Yaskawa INFORM job: DPRINT3D15.JBI

/JOB
//NAME DPRINT3D15
//POS
///NPOS 1161,0,0,0,0,0
///TOOL 9
///POSTYPE PULSE
///PULSE
C00000=36278,44575,-115468,79318,-120327,-85510,0
C00001=35662,44969,-114487,80045,-120135,-85172,0
C00002=36536,45454,-113310,79361,-120907,-84970,0
C00003=42251,40475,-125838,71885,-121337,-89052,0
C00004=39883,39258,-128907,73938,-119379,-89536,0
C00005=34290,44258,-116221,81147,-118965,-85469,0
C00006=35192,44719,-115096,80418,-119728,-85276,0
C00007=34956,44981,-114446,80729,-119702,-85074,0
C00008=35425,45232,-113838,80359,-120109,-84970,0
C00009=35608,45029,-114339,80116,-120129,-85126,0
C00010=36169,44682,-115203,79459,-120311,-85426,0
C00011=36133,44092,-116660,79301,-120005,-85809,0
C00012=40210,40493,-125752,74007,-120311,-88747,0
C00013=40210,40434,-125759,74020,-120337,-88719,0
C00014=36356,44563,-115373,79269,-120414,-85467,0
C00015=41022,40463,-125699,73192,-120772,-88813,0
C00016=40015,39945,-127000,74059,-119937,-89019,0
C00017=35392,44052,-116619,80042,-119585,-85678,0
C00018=36278,44521,-115476,79331,-120346,-85484,0
C00019=35662,44916,-114494,80057,-120153,-85146,0
C00020=36536,45401,-113317,79374,-120926,-84945,0
C00021=42251,40415,-125845,71899,-121365,-89025,0
C00022=39883,39197,-128913,73951,-119406,-89507,0
C00023=34290,44203,-116228,81159,-118982,-85443,0
C00024=35192,44665,-115103,80431,-119747,-85250,0
C00025=34956,44928,-114453,80742,-119720,-85049,0
C00026=35425,45178,-113845,80371,-120127,-84944,0
C00027=35608,44975,-114347,80129,-120148,-85100,0
C00028=36169,44628,-115210,79472,-120330,-85400,0
C00029=36133,44037,-116667,79314,-120025,-85783,0
C00030=40210,40434,-125759,74020,-120337,-88719,0
C00031=40211,40374,-125767,74034,-120363,-88691,0
C00032=36356,44509,-115380,79282,-120434,-85441,0
C00033=41022,40404,-125706,73206,-120798,-88785,0
C00034=40015,39885,-127008,74073,-119963,-88991,0
C00035=35393,43998,-116625,80054,-119604,-85652,0
C00036=36278,44467,-115483,79344,-120365,-85458,0
C00037=35663,44862,-114501,80070,-120172,-85120,0
C00038=36536,45348,-113324,79387,-120945,-84919,0
C00039=42252,40355,-125852,71914,-121393,-88997,0
C00040=39884,39135,-128921,73965,-119433,-89478,0
C00041=34290,44149,-116235,81171,-119001,-85416,0
C00042=35193,44611,-115110,80443,-119765,-85224,0
C00043=34957,44874,-114460,80754,-119739,-85022,0
C00044=35425,45125,-113852,80384,-120145,-84918,0
C00045=35608,44922,-114354,80141,-120166,-85074,0
C00046=36170,44574,-115218,79485,-120350,-85374,0
C00047=36133,43983,-116674,79327,-120044,-85756,0
C00048=40211,40374,-125767,74034,-120363,-88691,0
C00049=40211,40315,-125774,74048,-120389,-88662,0
C00050=36357,44456,-115387,79295,-120452,-85415,0
C00051=41022,40345,-125714,73220,-120825,-88758,0
C00052=40016,39824,-127015,74086,-119989,-88962,0
C00053=35393,43943,-116632,80066,-119622,-85625,0
C00054=36279,44413,-115490,79356,-120384,-85432,0
C00055=35663,44809,-114508,80082,-120190,-85094,0
C00056=36537,45295,-113331,79400,-120964,-84894,0
C00057=42252,40296,-125860,71928,-121421,-88969,0
C00058=39884,39074,-128928,73978,-119459,-89449,0
C00059=34291,44095,-116242,81183,-119019,-85390,0
C00060=35193,44558,-115117,80455,-119783,-85198,0
C00061=34957,44821,-114467,80766,-119756,-84996,0
C00062=35426,45072,-113859,80396,-120164,-84892,0
C00063=35609,44869,-114361,80154,-120184,-85048,0
C00064=36170,44520,-115225,79497,-120369,-85348,0
C00065=36134,43928,-116681,79339,-120064,-85730,0
C00066=40211,40315,-125774,74048,-120389,-88662,0
C00067=40212,40255,-125781,74062,-120414,-88635,0
C00068=36357,44402,-115394,79307,-120472,-85389,0
C00069=41023,40285,-125721,73234,-120851,-88730,0
C00070=40016,39764,-127022,74100,-120016,-88934,0
C00071=35393,43889,-116639,80079,-119642,-85599,0
C00072=36279,44359,-115497,79369,-120404,-85406,0
C00073=35663,44755,-114514,80095,-120210,-85068,0
C00074=36537,45242,-113338,79413,-120983,-84867,0
C00075=42253,40236,-125867,71943,-121449,-88942,0
C00076=39884,39012,-128936,73992,-119487,-89420,0
C00077=34291,44040,-116249,81195,-119038,-85364,0
C00078=35193,44504,-115124,80468,-119802,-85172,0
C00079=34958,44768,-114474,80779,-119774,-84970,0
C00080=35426,45019,-113866,80409,-120181,-84866,0
C00081=35609,44815,-114367,80167,-120203,-85022,0
C00082=36170,44467,-115232,79510,-120388,-85322,0
C00083=36134,43874,-116688,79352,-120084,-85704,0
C00084=40212,40255,-125781,74062,-120414,-88635,0
C00085=40212,40196,-125788,74075,-120441,-88607,0
C00086=36357,44348,-115400,79320,-120491,-85362,0
C00087=41023,40226,-125728,73248,-120877,-88702,0
C00088=40017,39704,-127030,74114,-120042,-88906,0
C00089=35394,43834,-116646,80091,-119660,-85573,0
C00090=36279,44305,-115503,79382,-120423,-85380,0
C00091=35664,44702,-114521,80108,-120228,-85042,0
C00092=36537,45189,-113344,79427,-121001,-84842,0
C00093=42253,40177,-125874,71957,-121476,-88914,0
C00094=39885,38951,-128943,74005,-119513,-89391,0
C00095=34291,43986,-116255,81207,-119055,-85337,0
C00096=35193,44450,-115130,80480,-119820,-85145,0
C00097=34958,44714,-114480,80791,-119793,-84945,0
C00098=35426,44966,-113872,80421,-120199,-84840,0
C00099=35609,44762,-114374,80179,-120221,-84996,0
C00100=36170,44413,-115237,79523,-120407,-85296,0
C00101=36134,43819,-116694,79365,-120104,-85677,0
C00102=40212,40196,-125788,74075,-120441,-88607,0
C00103=40212,40137,-125795,74089,-120466,-88578,0
C00104=36358,44294,-115406,79333,-120511,-85336,0
C00105=41024,40166,-125735,73263,-120904,-88674,0
C00106=40017,39644,-127037,74127,-120068,-88877,0
C00107=35394,43780,-116653,80104,-119680,-85546,0
C00108=36280,44251,-115510,79395,-120443,-85354,0
C00109=35664,44649,-114528,80121,-120246,-85016,0
C00110=36538,45136,-113351,79440,-121021,-84816,0
C00111=42253,40118,-125881,71971,-121504,-88886,0
C00112=39885,38889,-128950,74018,-119541,-89362,0
C00113=34292,43932,-116262,81219,-119073,-85311,0
C00114=35194,44397,-115137,80493,-119840,-85119,0
C00115=34958,44661,-114487,80803,-119811,-84919,0
C00116=35427,44913,-113879,80434,-120218,-84815,0
C00117=35610,44708,-114381,80192,-120241,-84970,0
C00118=36171,44359,-115244,79536,-120427,-85270,0
C00119=36135,43765,-116701,79378,-120124,-85651,0
C00120=40212,40137,-125795,74089,-120466,-88578,0
C00121=40213,40077,-125802,74103,-120492,-88550,0
C00122=36358,44240,-115413,79346,-120530,-85310,0
C00123=41024,40107,-125742,73277,-120931,-88646,0
C00124=40017,39584,-127044,74141,-120095,-88849,0
C00125=35394,43726,-116659,80116,-119699,-85520,0
C00126=36280,44198,-115517,79408,-120463,-85328,0
C00127=35664,44595,-114534,80133,-120265,-84990,0
C00128=36538,45083,-113358,79453,-121039,-84791,0
C00129=42254,40058,-125888,71986,-121531,-88859,0
C00130=39886,38828,-128957,74032,-119567,-89333,0
C00131=34292,43878,-116269,81231,-119092,-85284,0
C00132=35194,44343,-115144,80505,-119858,-85093,0
C00133=34958,44607,-114494,80816,-119829,-84892,0
C00134=35427,44860,-113885,80447,-120236,-84789,0
C00135=35610,44655,-114387,80205,-120259,-84944,0
C00136=36171,44305,-115251,79549,-120446,-85243,0
C00137=36135,43711,-116708,79391,-120143,-85624,0
C00138=40213,40077,-125802,74103,-120492,-88550,0
C00139=40213,40018,-125808,74117,-120519,-88522,0
C00140=36358,44187,-115420,79359,-120550,-85284,0
C00141=41024,40048,-125749,73291,-120958,-88618,0
C00142=40018,39524,-127051,74155,-120120,-88820,0
C00143=35395,43671,-116666,80129,-119718,-85493,0
C00144=36280,44144,-115523,79421,-120482,-85302,0
C00145=35664,44542,-114541,80146,-120284,-84964,0
C00146=36538,45031,-113364,79466,-121059,-84765,0
C00147=42254,39999,-125895,72001,-121559,-88831,0
C00148=39886,38767,-128964,74046,-119595,-89304,0
C00149=34292,43824,-116275,81243,-119110,-85257,0
C00150=35194,44289,-115150,80518,-119876,-85067,0
C00151=34959,44554,-114500,80828,-119847,-84866,0
C00152=35427,44807,-113892,80460,-120255,-84762,0
C00153=35610,44602,-114394,80218,-120278,-84918,0
C00154=36171,44252,-115258,79562,-120465,-85217,0
C00155=36135,43656,-116714,79403,-120163,-85597,0
C00156=40213,40018,-125808,74117,-120519,-88522,0
C00157=40214,39959,-125815,74131,-120544,-88494,0
C00158=36359,44133,-115426,79373,-120569,-85257,0
C00159=41025,39989,-125756,73305,-120984,-88590,0
C00160=40018,39464,-127058,74168,-120147,-88792,0
C00161=35395,43617,-116673,80142,-119737,-85466,0
C00162=36281,44090,-115529,79434,-120500,-85275,0
C00163=35665,44489,-114547,80159,-120303,-84938,0
C00164=36539,44978,-113371,79479,-121077,-84739,0
C00165=42255,39939,-125901,72015,-121586,-88803,0
C00166=39886,38705,-128971,74059,-119621,-89275,0
C00167=34293,43770,-116282,81255,-119127,-85231,0
C00168=35195,44236,-115157,80531,-119895,-85041,0
C00169=34959,44501,-114507,80841,-119865,-84840,0
C00170=35428,44754,-113898,80472,-120273,-84737,0
C00171=35611,44549,-114400,80230,-120296,-84892,0
C00172=36172,44198,-115264,79575,-120484,-85191,0
C00173=36136,43602,-116721,79416,-120182,-85571,0
C00174=40214,39959,-125815,74131,-120544,-88494,0
C00175=40214,39899,-125822,74145,-120571,-88466,0
C00176=36359,44079,-115433,79386,-120589,-85231,0
C00177=41025,39929,-125761,73319,-121011,-88562,0
C00178=40019,39403,-127063,74182,-120173,-88763,0
C00179=35395,43563,-116678,80154,-119756,-85440,0
C00180=36281,44036,-115536,79447,-120520,-85249,0
C00181=35665,44435,-114554,80172,-120321,-84912,0
C00182=36539,44925,-113377,79492,-121097,-84713,0
C00183=42255,39880,-125908,72030,-121614,-88775,0
C00184=39887,38644,-128978,74073,-119649,-89246,0
C00185=34293,43716,-116288,81267,-119146,-85205,0
C00186=35195,44182,-115163,80543,-119913,-85014,0
C00187=34959,44448,-114513,80853,-119883,-84814,0
C00188=35428,44701,-113905,80485,-120291,-84711,0
C00189=35611,44496,-114407,80243,-120314,-84866,0
C00190=36172,44145,-115271,79588,-120504,-85165,0
C00191=36136,43548,-116728,79429,-120202,-85545,0
C00192=40214,39899,-125822,74145,-120571,-88466,0
C00193=40214,39840,-125829,74159,-120596,-88438,0
C00194=36359,44026,-115438,79399,-120608,-85205,0
C00195=41026,39870,-125768,73334,-121037,-88534,0
C00196=40019,39343,-127070,74196,-120199,-88735,0
C00197=35396,43509,-116685,80167,-119775,-85413,0
C00198=36281,43983,-115542,79460,-120540,-85223,0
C00199=35666,44382,-114560,80185,-120340,-84885,0
C00200=36539,44872,-113383,79506,-121115,-84688,0
C00201=42256,39821,-125914,72044,-121642,-88747,0
C00202=39887,38583,-128985,74087,-119675,-89217,0
C00203=34293,43662,-116295,81279,-119164,-85178,0
C00204=35195,44129,-115170,80556,-119932,-84988,0
C00205=34960,44394,-114519,80866,-119902,-84787,0
C00206=35428,44648,-113911,80498,-120310,-84685,0
C00207=35611,44442,-114413,80256,-120334,-84840,0
C00208=36172,44091,-115276,79601,-120523,-85138,0
C00209=36136,43493,-116734,79442,-120221,-85518,0
C00210=40214,39840,-125829,74159,-120596,-88438,0
C00211=40215,39781,-125835,74173,-120622,-88409,0
C00212=36360,43972,-115445,79412,-120628,-85179,0
C00213=41026,39811,-125775,73348,-121065,-88506,0
C00214=40019,39284,-127077,74210,-120226,-88706,0
C00215=35396,43454,-116691,80180,-119795,-85386,0
C00216=36282,43929,-115549,79473,-120559,-85196,0
C00217=35666,44329,-114566,80197,-120359,-84859,0
C00218=36540,44820,-113389,79519,-121135,-84661,0
C00219=42256,39762,-125921,72059,-121670,-88719,0
C00220=39888,38522,-128990,74100,-119703,-89188,0
C00221=34294,43608,-116300,81292,-119182,-85151,0
C00222=35196,44075,-115175,80568,-119950,-84962,0
C00223=34960,44341,-114525,80878,-119920,-84761,0
C00224=35429,44595,-113917,80511,-120328,-84659,0
C00225=35612,44389,-114419,80269,-120352,-84814,0
C00226=36173,44038,-115283,79614,-120542,-85112,0
C00227=36137,43439,-116739,79455,-120241,-85491,0
C00228=40215,39781,-125835,74173,-120622,-88409,0
C00229=40215,39722,-125842,74187,-120649,-88381,0
C00230=36360,43919,-115451,79425,-120648,-85152,0
C00231=41027,39752,-125781,73362,-121091,-88478,0
C00232=40020,39224,-127083,74224,-120252,-88678,0
C00233=35396,43400,-116697,80192,-119813,-85360,0
C00234=36282,43876,-115554,79487,-120579,-85170,0
C00235=35666,44276,-114572,80210,-120377,-84833,0
C00236=36540,44767,-113395,79532,-121153,-84635,0
C00237=42256,39702,-125928,72074,-121698,-88691,0
C00238=39888,38460,-128997,74114,-119729,-89159,0
C00239=34294,43554,-116307,81304,-119201,-85125,0
C00240=35196,44022,-115181,80581,-119968,-84935,0
C00241=34960,44288,-114532,80891,-119937,-84735,0
C00242=35429,44542,-113923,80523,-120346,-84632,0
C00243=35612,44336,-114425,80282,-120371,-84787,0
C00244=36173,43984,-115289,79627,-120561,-85086,0
C00245=36137,43385,-116746,79468,-120260,-85465,0
C00246=40215,39722,-125842,74187,-120649,-88381,0
C00247=40216,39663,-125847,74201,-120674,-88353,0
C00248=36360,43865,-115457,79438,-120667,-85126,0
C00249=41027,39693,-125788,73377,-121118,-88449,0
C00250=40020,39164,-127090,74238,-120279,-88649,0
C00251=35397,43346,-116704,80205,-119833,-85333,0
C00252=36282,43822,-115560,79500,-120598,-85143,0
C00253=35667,44223,-114578,80223,-120396,-84807,0
C00254=36540,44715,-113401,79546,-121173,-84610,0
C00255=42257,39643,-125934,72089,-121725,-88663,0
C00256=39889,38399,-129004,74128,-119757,-89130,0
C00257=34294,43500,-116313,81316,-119218,-85098,0
C00258=35196,43969,-115188,80594,-119987,-84909,0
C00259=34961,44235,-114537,80904,-119956,-84709,0
C00260=35429,44489,-113929,80536,-120365,-84606,0
C00261=35612,44283,-114431,80295,-120389,-84761,0
C00262=36174,43931,-115295,79640,-120581,-85060,0
C00263=36137,43331,-116752,79481,-120280,-85438,0
C00264=40216,39663,-125847,74201,-120674,-88353,0
C00265=40216,39604,-125854,74215,-120700,-88325,0
C00266=36361,43811,-115463,79451,-120687,-85100,0
C00267=41027,39634,-125793,73391,-121144,-88421,0
C00268=40021,39104,-127095,74252,-120305,-88620,0
C00269=35397,43292,-116709,80218,-119852,-85306,0
C00270=36283,43768,-115566,79513,-120618,-85117,0
C00271=35667,44170,-114584,80236,-120415,-84780,0
C00272=36541,44662,-113407,79559,-121192,-84584,0
C00273=42257,39584,-125939,72104,-121753,-88635,0
C00274=39889,38338,-129010,74142,-119783,-89100,0
C00275=34294,43446,-116319,81328,-119236,-85071,0
C00276=35197,43915,-115194,80607,-120006,-84883,0
C00277=34961,44182,-114543,80916,-119974,-84682,0
C00278=35430,44436,-113935,80549,-120383,-84580,0
C00279=35613,44230,-114437,80308,-120407,-84735,0
C00280=36174,43877,-115301,79653,-120600,-85033,0
C00281=36138,43277,-116758,79494,-120300,-85411,0
C00282=40216,39604,-125854,74215,-120700,-88325,0
C00283=40216,39545,-125860,74229,-120727,-88296,0
C00284=36361,43758,-115469,79465,-120705,-85073,0
C00285=41028,39575,-125799,73406,-121170,-88393,0
C00286=40021,39044,-127102,74266,-120332,-88592,0
C00287=35397,43238,-116715,80231,-119871,-85279,0
C00288=36283,43715,-115572,79526,-120637,-85090,0
C00289=35667,44117,-114590,80249,-120434,-84754,0
C00290=36541,44609,-113413,79573,-121211,-84558,0
C00291=42258,39525,-125946,72118,-121781,-88607,0
C00292=39889,38277,-129017,74155,-119811,-89071,0
C00293=34295,43392,-116324,81341,-119255,-85044,0
C00294=35197,43862,-115199,80619,-120025,-84856,0
C00295=34961,44129,-114549,80929,-119993,-84656,0
C00296=35430,44384,-113941,80562,-120402,-84554,0
C00297=35613,44177,-114443,80321,-120427,-84709,0
C00298=36174,43824,-115306,79667,-120620,-85007,0
C00299=36138,43223,-116763,79508,-120320,-85384,0
C00300=40216,39545,-125860,74229,-120727,-88296,0
C00301=40217,39485,-125866,74244,-120752,-88268,0
C00302=36361,43705,-115475,79478,-120725,-85047,0
C00303=41028,39516,-125806,73420,-121198,-88365,0
C00304=40022,38984,-127108,74280,-120358,-88563,0
C00305=35398,43184,-116721,80243,-119890,-85253,0
C00306=36283,43661,-115579,79539,-120657,-85064,0
C00307=35667,44064,-114596,80262,-120452,-84728,0
C00308=36541,44557,-113419,79586,-121230,-84532,0
C00309=42258,39466,-125952,72133,-121809,-88579,0
C00310=39890,38216,-129023,74169,-119837,-89041,0
C00311=34295,43338,-116330,81353,-119273,-85018,0
C00312=35197,43808,-115205,80632,-120043,-84830,0
C00313=34962,44076,-114555,80942,-120011,-84630,0
C00314=35430,44331,-113947,80575,-120420,-84528,0
C00315=35613,44124,-114449,80334,-120445,-84682,0
C00316=36175,43770,-115312,79680,-120638,-84981,0
C00317=36138,43169,-116769,79521,-120340,-85358,0
C00318=40217,39485,-125866,74244,-120752,-88268,0
C00319=40217,39426,-125872,74258,-120779,-88239,0
C00320=36362,43651,-115481,79491,-120744,-85021,0
C00321=41029,39457,-125812,73435,-121224,-88336,0
C00322=40022,38924,-127114,74294,-120384,-88534,0
C00323=35398,43130,-116727,80256,-119909,-85226,0
C00324=36284,43608,-115583,79553,-120676,-85037,0
C00325=35668,44011,-114601,80275,-120472,-84702,0
C00326=36542,44504,-113424,79600,-121249,-84505,0
C00327=42259,39407,-125958,72148,-121837,-88550,0
C00328=39890,38155,-129028,74183,-119865,-89012,0
C00329=34296,43284,-116336,81365,-119292,-84990,0
C00330=35198,43755,-115211,80645,-120061,-84803,0
C00331=34962,44023,-114561,80955,-120029,-84603,0
C00332=35431,44278,-113952,80588,-120438,-84501,0
C00333=35614,44071,-114454,80347,-120464,-84656,0
C00334=36175,43717,-115318,79693,-120658,-84954,0
C00335=36139,43115,-116775,79534,-120359,-85331,0
C00336=40217,39426,-125872,74258,-120779,-88239,0
C00337=40218,39367,-125877,74272,-120805,-88211,0
C00338=36362,43598,-115486,79505,-120764,-84994,0
C00339=41029,39398,-125818,73449,-121251,-88308,0
C00340=40022,38864,-127120,74308,-120411,-88505,0
C00341=35398,43076,-116732,80269,-119928,-85199,0
C00342=36284,43554,-115589,79566,-120696,-85011,0
C00343=35668,43958,-114607,80288,-120490,-84675,0
C00344=36542,44452,-113430,79613,-121268,-84480,0
C00345=42259,39348,-125964,72163,-121864,-88523,0
C00346=39891,38094,-129034,74197,-119891,-88983,0
C00347=34296,43230,-116342,81378,-119309,-84964,0
C00348=35198,43702,-115217,80658,-120080,-84776,0
C00349=34962,43970,-114566,80967,-120047,-84577,0
C00350=35431,44225,-113958,80601,-120457,-84475,0
C00351=35614,44018,-114460,80360,-120482,-84630,0
C00352=36175,43664,-115324,79706,-120677,-84927,0
C00353=36139,43061,-116781,79547,-120379,-85304,0
C00354=40218,39367,-125877,74272,-120805,-88211,0
C00355=40218,39308,-125883,74287,-120830,-88183,0
C00356=36362,43544,-115491,79518,-120783,-84967,0
C00357=41029,39339,-125823,73464,-121277,-88280,0
C00358=40023,38805,-127125,74323,-120437,-88476,0
C00359=35399,43022,-116738,80282,-119948,-85172,0
C00360=36284,43501,-115595,79579,-120715,-84984,0
C00361=35668,43905,-114612,80302,-120508,-84649,0
C00362=36542,44400,-113436,79627,-121286,-84454,0
C00363=42259,39289,-125969,72178,-121892,-88494,0
C00364=39891,38033,-129040,74211,-119919,-88954,0
C00365=34296,43177,-116347,81390,-119327,-84937,0
C00366=35198,43649,-115222,80671,-120098,-84750,0
C00367=34963,43917,-114572,80980,-120065,-84551,0
C00368=35431,44173,-113963,80614,-120475,-84449,0
C00369=35614,43965,-114465,80373,-120502,-84603,0
C00370=36175,43611,-115329,79720,-120697,-84901,0
C00371=36140,43007,-116786,79560,-120398,-85278,0
C00372=40218,39308,-125883,74287,-120830,-88183,0
C00373=40218,39250,-125889,74301,-120857,-88154,0
C00374=36363,43491,-115497,79531,-120803,-84941,0
C00375=41030,39280,-125829,73479,-121305,-88252,0
C00376=40023,38745,-127131,74337,-120464,-88447,0
C00377=35399,42968,-116744,80295,-119966,-85145,0
C00378=36285,43448,-115600,79593,-120735,-84958,0
C00379=35669,43852,-114618,80315,-120528,-84623,0
C00380=36543,44347,-113441,79640,-121306,-84428,0
C00381=42260,39230,-125975,72194,-121920,-88466,0
C00382=39891,37972,-129047,74225,-119945,-88924,0
C00383=34296,43123,-116353,81403,-119346,-84910,0
C00384=35199,43595,-115227,80684,-120117,-84724,0
C00385=34963,43864,-114577,80993,-120083,-84524,0
C00386=35432,44120,-113969,80627,-120494,-84423,0
C00387=35615,43913,-114471,80386,-120520,-84577,0
C00388=36176,43557,-115335,79733,-120716,-84874,0
C00389=36140,42953,-116792,79574,-120419,-85250,0
C00390=40218,39250,-125889,74301,-120857,-88154,0
C00391=40219,39191,-125895,74315,-120883,-88125,0
C00392=36363,43438,-115503,79545,-120822,-84914,0
C00393=41030,39221,-125835,73493,-121331,-88223,0
C00394=40024,38685,-127137,74351,-120490,-88418,0
C00395=35399,42914,-116748,80308,-119986,-85119,0
C00396=36285,43394,-115606,79606,-120754,-84931,0
C00397=35669,43799,-114623,80328,-120546,-84596,0
C00398=36543,44295,-113446,79654,-121326,-84401,0
C00399=42260,39171,-125981,72209,-121948,-88438,0
C00400=39892,37911,-129051,74239,-119973,-88895,0
C00401=34297,43069,-116358,81415,-119364,-84883,0
C00402=35199,43542,-115233,80697,-120136,-84697,0
C00403=34963,43811,-114583,81006,-120102,-84498,0
C00404=35432,44068,-113974,80640,-120512,-84396,0
C00405=35615,43860,-114476,80399,-120538,-84551,0
C00406=36176,43504,-115340,79746,-120735,-84848,0
C00407=36140,42899,-116798,79587,-120438,-85224,0
C00408=40219,39191,-125895,74315,-120883,-88125,0
C00409=40219,39132,-125900,74330,-120910,-88097,0
C00410=36363,43385,-115507,79558,-120842,-84888,0
C00411=41031,39162,-125841,73508,-121358,-88195,0
C00412=40024,38626,-127143,74365,-120517,-88390,0
C00413=35400,42860,-116754,80321,-120005,-85091,0
C00414=36285,43341,-115611,79619,-120774,-84905,0
C00415=35669,43746,-114628,80341,-120565,-84570,0
C00416=36543,44243,-113452,79668,-121344,-84375,0
C00417=42261,39112,-125987,72224,-121976,-88409,0
C00418=39892,37850,-129057,74254,-120001,-88865,0
C00419=34297,43016,-116363,81428,-119382,-84856,0
C00420=35199,43489,-115238,80710,-120155,-84670,0
C00421=34964,43758,-114588,81019,-120120,-84471,0
C00422=35432,44015,-113979,80653,-120530,-84370,0
C00423=35615,43807,-114481,80412,-120557,-84525,0
C00424=36176,43451,-115345,79760,-120754,-84821,0
C00425=36141,42845,-116802,79600,-120458,-85197,0
C00426=40219,39132,-125900,74330,-120910,-88097,0
C00427=40220,39073,-125906,74344,-120935,-88068,0
C00428=36364,43331,-115513,79572,-120861,-84861,0
C00429=41031,39103,-125845,73523,-121385,-88166,0
C00430=40024,38566,-127148,74380,-120543,-88361,0
C00431=35400,42806,-116759,80334,-120024,-85065,0
C00432=36286,43288,-115617,79633,-120793,-84878,0
C00433=35670,43693,-114634,80354,-120584,-84543,0
C00434=36544,44190,-113457,79681,-121363,-84349,0
C00435=42261,39053,-125992,72239,-122004,-88381,0
C00436=39893,37789,-129063,74268,-120027,-88835,0
C00437=34297,42962,-116368,81440,-119401,-84829,0
C00438=35200,43436,-115243,80723,-120173,-84643,0
C00439=34964,43706,-114593,81032,-120138,-84444,0
C00440=35433,43963,-113985,80666,-120549,-84344,0
C00441=35616,43754,-114487,80425,-120576,-84498,0
C00442=36177,43398,-115351,79773,-120774,-84795,0
C00443=36141,42791,-116808,79613,-120477,-85170,0
C00444=40220,39073,-125906,74344,-120935,-88068,0
C00445=40220,39014,-125911,74359,-120961,-88039,0
C00446=36364,43278,-115518,79585,-120881,-84834,0
C00447=41031,39045,-125851,73538,-121412,-88138,0
C00448=40025,38506,-127153,74394,-120569,-88332,0
C00449=35400,42753,-116765,80347,-120043,-85037,0
C00450=36286,43235,-115621,79646,-120813,-84851,0
C00451=35670,43640,-114639,80368,-120603,-84516,0
C00452=36544,44138,-113462,79695,-121383,-84323,0
C00453=42262,38994,-125997,72254,-122032,-88353,0
C00454=39893,37728,-129069,74282,-120055,-88806,0
C00455=34298,42908,-116374,81453,-119419,-84802,0
C00456=35200,43383,-115248,80736,-120191,-84617,0
C00457=34964,43653,-114598,81045,-120157,-84418,0
C00458=35433,43910,-113990,80680,-120567,-84317,0
C00459=35616,43702,-114492,80439,-120595,-84471,0
C00460=36177,43345,-115356,79787,-120793,-84768,0
C00461=36141,42737,-116813,79627,-120497,-85143,0
C00462=40220,39014,-125911,74359,-120961,-88039,0
C00463=40220,38955,-125916,74374,-120988,-88011,0
C00464=36364,43225,-115523,79599,-120900,-84808,0
C00465=41032,38986,-125857,73553,-121438,-88109,0
C00466=40025,38447,-127159,74409,-120596,-88303,0
C00467=35401,42699,-116769,80360,-120063,-85010,0
C00468=36286,43181,-115627,79660,-120833,-84825,0
C00469=35670,43588,-114644,80381,-120621,-84490,0
C00470=36544,44086,-113467,79709,-121401,-84296,0
C00471=42262,38935,-126003,72269,-122060,-88325,0
C00472=39894,37668,-129074,74296,-120081,-88776,0
C00473=34298,42855,-116378,81465,-119436,-84775,0
C00474=35200,43330,-115253,80749,-120210,-84590,0
C00475=34965,43600,-114603,81058,-120175,-84391,0
C00476=35433,43858,-113995,80693,-120585,-84291,0
C00477=35616,43649,-114497,80452,-120613,-84444,0
C00478=36178,43292,-115360,79800,-120813,-84742,0
C00479=36142,42684,-116819,79640,-120517,-85116,0
C00480=40220,38955,-125916,74374,-120988,-88011,0
C00481=40221,38897,-125921,74388,-121014,-87982,0
C00482=36365,43172,-115528,79613,-120920,-84781,0
C00483=41032,38927,-125861,73568,-121466,-88080,0
C00484=40026,38388,-127163,74423,-120622,-88274,0
C00485=35401,42645,-116775,80373,-120082,-84984,0
C00486=36287,43128,-115631,79673,-120852,-84798,0
C00487=35671,43535,-114649,80394,-120641,-84464,0
C00488=36545,44034,-113472,79722,-121421,-84270,0
C00489=42262,38876,-126007,72285,-122087,-88296,0
C00490=39894,37607,-129079,74310,-120109,-88747,0
C00491=34298,42801,-116384,81478,-119455,-84748,0
C00492=35201,43277,-115258,80762,-120229,-84563,0
C00493=34965,43547,-114608,81071,-120192,-84365,0
C00494=35434,43805,-114000,80706,-120604,-84265,0
C00495=35617,43596,-114502,80465,-120633,-84418,0
C00496=36178,43239,-115366,79814,-120833,-84715,0
C00497=36142,42630,-116823,79654,-120537,-85089,0
C00498=40221,38897,-125921,74388,-121014,-87982,0
C00499=40221,38838,-125927,74403,-121039,-87953,0
C00500=36365,43119,-115533,79626,-120939,-84754,0
C00501=41033,38869,-125866,73582,-121492,-88052,0
C00502=40026,38328,-127169,74437,-120649,-88244,0
C00503=35401,42592,-116779,80386,-120101,-84956,0
C00504=36287,43075,-115636,79687,-120872,-84771,0
C00505=35671,43482,-114654,80407,-120659,-84437,0
C00506=36545,43982,-113476,79736,-121439,-84244,0
C00507=42263,38818,-126013,72300,-122115,-88268,0
C00508=39894,37546,-129085,74325,-120136,-88717,0
C00509=34299,42748,-116389,81491,-119473,-84721,0
C00510=35201,43224,-115263,80775,-120248,-84537,0
C00511=34965,43495,-114613,81083,-120211,-84338,0
C00512=35434,43753,-114005,80719,-120622,-84238,0
C00513=35617,43544,-114506,80479,-120651,-84392,0
C00514=36178,43185,-115371,79827,-120852,-84688,0
C00515=36142,42576,-116828,79667,-120557,-85062,0
C00516=40221,38838,-125927,74403,-121039,-87953,0
C00517=40222,38779,-125931,74417,-121066,-87924,0
C00518=36365,43066,-115537,79640,-120959,-84728,0
C00519=41033,38810,-125872,73598,-121519,-88024,0
C00520=40026,38269,-127174,74452,-120675,-88215,0
C00521=35402,42538,-116784,80400,-120120,-84929,0
C00522=36287,43022,-115641,79701,-120891,-84744,0
C00523=35671,43430,-114658,80421,-120677,-84410,0
C00524=36545,43929,-113481,79750,-121459,-84218,0
C00525=42263,38759,-126018,72316,-122144,-88239,0
C00526=39895,37485,-129089,74339,-120163,-88687,0
C00527=34299,42694,-116393,81503,-119491,-84694,0
C00528=35201,43171,-115268,80788,-120266,-84510,0
C00529=34966,43442,-114618,81097,-120229,-84312,0
C00530=35434,43700,-114009,80733,-120641,-84211,0
C00531=35617,43491,-114511,80492,-120669,-84365,0
C00532=36179,43132,-115375,79841,-120870,-84661,0
C00533=36143,42522,-116832,79681,-120576,-85035,0
C00534=40222,38779,-125931,74417,-121066,-87924,0
C00535=40222,38721,-125936,74432,-121092,-87896,0
C00536=36366,43013,-115542,79653,-120980,-84701,0
C00537=41034,38751,-125876,73612,-121546,-87995,0
C00538=40027,38209,-127179,74467,-120702,-88186,0
C00539=35402,42484,-116789,80413,-120140,-84902,0
C00540=36288,42969,-115645,79714,-120911,-84717,0
C00541=35672,43377,-114663,80434,-120697,-84384,0
C00542=36546,43877,-113486,79764,-121478,-84191,0
C00543=42264,38700,-126022,72331,-122171,-88211,0
C00544=39895,37425,-129094,74354,-120190,-88658,0
C00545=34299,42641,-116398,81516,-119510,-84667,0
C00546=35202,43118,-115273,80801,-120284,-84483,0
C00547=34966,43390,-114622,81110,-120248,-84285,0
C00548=35434,43648,-114014,80746,-120660,-84185,0
C00549=35618,43438,-114516,80505,-120688,-84338,0
C00550=36179,43079,-115380,79854,-120890,-84634,0
C00551=36143,42469,-116837,79694,-120596,-85008,0
C00552=40222,38721,-125936,74432,-121092,-87896,0
C00553=40223,38662,-125942,74447,-121119,-87867,0
C00554=36366,42960,-115546,79667,-120999,-84674,0
C00555=41034,38693,-125881,73628,-121573,-87966,0
C00556=40027,38150,-127184,74481,-120728,-88157,0
C00557=35402,42431,-116793,80426,-120158,-84875,0
C00558=36288,42916,-115650,79728,-120930,-84691,0
C00559=35672,43324,-114668,80448,-120715,-84357,0
C00560=36546,43825,-113490,79778,-121497,-84165,0
C00561=42264,38642,-126028,72346,-122199,-88182,0
C00562=39896,37364,-129100,74368,-120218,-88628,0
C00563=34300,42587,-116403,81529,-119528,-84639,0
C00564=35202,43065,-115278,80814,-120303,-84456,0
C00565=34966,43337,-114627,81123,-120266,-84258,0
C00566=35435,43596,-114019,80759,-120679,-84158,0
C00567=35618,43386,-114520,80519,-120707,-84312,0
C00568=36179,43027,-115384,79868,-120910,-84608,0
C00569=36143,42415,-116842,79708,-120617,-84981,0
C00570=40223,38662,-125942,74447,-121119,-87867,0
C00571=40223,38604,-125946,74462,-121145,-87838,0
C00572=36366,42907,-115551,79681,-121019,-84647,0
C00573=41034,38634,-125885,73643,-121600,-87937,0
C00574=40028,38090,-127189,74496,-120754,-88127,0
C00575=35403,42377,-116798,80439,-120178,-84848,0
C00576=36288,42863,-115654,79742,-120950,-84664,0
C00577=35672,43272,-114672,80461,-120734,-84330,0
C00578=36546,43773,-113495,79792,-121516,-84138,0
C00579=42264,38583,-126032,72362,-122228,-88154,0
C00580=39896,37303,-129104,74383,-120244,-88598,0
C00581=34300,42534,-116407,81542,-119547,-84612,0
C00582=35202,43013,-115282,80827,-120322,-84429,0
C00583=34967,43284,-114631,81136,-120284,-84231,0
C00584=35435,43544,-114023,80773,-120697,-84132,0
C00585=35618,43333,-114525,80532,-120726,-84285,0
C00586=36179,42974,-115389,79882,-120929,-84581,0
C00587=36144,42362,-116846,79721,-120636,-84953,0
C00588=40223,38604,-125946,74462,-121145,-87838,0
C00589=40223,38545,-125951,74477,-121170,-87809,0
C00590=36367,42854,-115556,79695,-121038,-84620,0
C00591=41035,38576,-125890,73658,-121627,-87909,0
C00592=40028,38031,-127193,74511,-120781,-88098,0
C00593=35403,42324,-116802,80452,-120197,-84820,0
C00594=36289,42810,-115659,79755,-120969,-84637,0
C00595=35673,43219,-114677,80475,-120753,-84303,0
C00596=36547,43721,-113499,79805,-121536,-84112,0
C00597=42265,38524,-126037,72378,-122255,-88125,0
C00598=39896,37243,-129109,74397,-120272,-88568,0
C00599=34300,42481,-116412,81554,-119565,-84585,0
C00600=35203,42960,-115286,80841,-120341,-84402,0
C00601=34967,43232,-114636,81149,-120303,-84204,0
C00602=35436,43491,-114027,80786,-120715,-84105,0
C00603=35619,43281,-114529,80546,-120744,-84258,0
C00604=36180,42921,-115394,79895,-120949,-84554,0
C00605=36144,42308,-116851,79735,-120656,-84927,0
C00606=40223,38545,-125951,74477,-121170,-87809,0
C00607=40224,38487,-125955,74491,-121197,-87780,0
C00608=36367,42801,-115560,79709,-121058,-84593,0
C00609=41035,38517,-125895,73673,-121653,-87880,0
C00610=40028,37972,-127198,74525,-120807,-88069,0
C00611=35403,42270,-116807,80466,-120217,-84793,0
C00612=36289,42757,-115664,79769,-120989,-84610,0
C00613=35673,43167,-114681,80488,-120772,-84277,0
C00614=36547,43669,-113504,79819,-121554,-84085,0
C00615=42265,38466,-126042,72393,-122284,-88097,0
C00616=39897,37182,-129113,74412,-120299,-88539,0
C00617=34301,42427,-116416,81567,-119583,-84558,0
C00618=35203,42907,-115290,80854,-120359,-84375,0
C00619=34967,43180,-114640,81162,-120321,-84178,0
C00620=35436,43439,-114032,80799,-120734,-84078,0
C00621=35619,43229,-114534,80559,-120764,-84232,0
C00622=36180,42868,-115398,79909,-120968,-84527,0
C00623=36144,42255,-116855,79749,-120675,-84899,0
C00624=40224,38487,-125955,74491,-121197,-87780,0
C00625=40224,38428,-125960,74506,-121223,-87751,0
C00626=36367,42748,-115565,79722,-121077,-84566,0
C00627=41036,38459,-125899,73688,-121681,-87851,0
C00628=40029,37912,-127202,74540,-120834,-88040,0
C00629=35404,42217,-116812,80479,-120235,-84766,0
C00630=36289,42704,-115668,79783,-121008,-84583,0
C00631=35673,43114,-114685,80502,-120791,-84249,0
C00632=36547,43617,-113508,79833,-121574,-84059,0
C00633=42266,38407,-126046,72409,-122312,-88068,0
C00634=39897,37122,-129118,74426,-120326,-88509,0
C00635=34301,42374,-116420,81580,-119601,-84531,0
C00636=35203,42854,-115295,80867,-120377,-84349,0
C00637=34967,43127,-114645,81175,-120340,-84151,0
C00638=35436,43387,-114036,80813,-120752,-84052,0
C00639=35619,43176,-114538,80573,-120782,-84205,0
C00640=36180,42815,-115402,79923,-120988,-84500,0
C00641=36145,42201,-116860,79762,-120695,-84872,0
C00642=40224,38428,-125960,74506,-121223,-87751,0
C00643=40225,38370,-125964,74521,-121250,-87722,0
C00644=36368,42695,-115568,79736,-121097,-84539,0
C00645=41036,38400,-125904,73704,-121707,-87822,0
C00646=40029,37853,-127207,74555,-120861,-88011,0
C00647=35404,42163,-116815,80492,-120255,-84739,0
C00648=36290,42651,-115672,79797,-121028,-84556,0
C00649=35674,43062,-114689,80515,-120810,-84223,0
C00650=36548,43566,-113512,79847,-121593,-84032,0
C00651=42266,38349,-126050,72424,-122339,-88039,0
C00652=39898,37061,-129123,74441,-120353,-88479,0
C00653=34301,42321,-116424,81593,-119619,-84504,0
C00654=35204,42801,-115299,80881,-120397,-84321,0
C00655=34968,43075,-114649,81189,-120358,-84124,0
C00656=35436,43335,-114040,80826,-120771,-84025,0
C00657=35620,43124,-114542,80586,-120800,-84178,0
C00658=36181,42762,-115406,79937,-121007,-84473,0
C00659=36145,42148,-116863,79776,-120715,-84845,0
C00660=40225,38370,-125964,74521,-121250,-87722,0
C00661=40225,38311,-125968,74536,-121276,-87693,0
C00662=36368,42642,-115573,79750,-121116,-84512,0
C00663=41036,38342,-125908,73719,-121735,-87793,0
C00664=40030,37794,-127212,74570,-120888,-87981,0
C00665=35404,42110,-116820,80506,-120274,-84711,0
C00666=36290,42598,-115676,79811,-121047,-84529,0
C00667=35674,43010,-114694,80529,-120828,-84196,0
C00668=36548,43514,-113516,79861,-121612,-84006,0
C00669=42267,38290,-126054,72440,-122368,-88010,0
C00670=39898,37001,-129127,74456,-120381,-88449,0
C00671=34302,42268,-116429,81606,-119637,-84476,0
C00672=35204,42749,-115303,80894,-120415,-84294,0
C00673=34968,43022,-114653,81202,-120376,-84097,0
C00674=35437,43283,-114044,80840,-120789,-83998,0
C00675=35620,43071,-114546,80600,-120820,-84151,0
C00676=36181,42710,-115411,79950,-121027,-84446,0
C00677=36145,42094,-116868,79790,-120735,-84818,0
C00678=40225,38311,-125968,74536,-121276,-87693,0
C00679=40225,38253,-125973,74551,-121303,-87664,0
C00680=36368,42590,-115576,79764,-121136,-84485,0
C00681=41037,38284,-125912,73734,-121761,-87764,0
C00682=40030,37735,-127215,74585,-120914,-87952,0
C00683=35405,42056,-116823,80519,-120294,-84684,0
C00684=36290,42545,-115680,79824,-121067,-84502,0
C00685=35674,42957,-114698,80542,-120847,-84169,0
C00686=36548,43462,-113520,79876,-121631,-83979,0
C00687=42267,38232,-126059,72456,-122395,-87982,0
C00688=39899,36940,-129131,74470,-120409,-88419,0
C00689=34302,42215,-116432,81619,-119656,-84449,0
C00690=35204,42696,-115307,80907,-120434,-84267,0
C00691=34968,42970,-114657,81215,-120395,-84070,0
C00692=35437,43231,-114048,80853,-120807,-83972,0
C00693=35620,43019,-114550,80613,-120838,-84124,0
C00694=36182,42657,-115414,79964,-121046,-84420,0
C00695=36146,42041,-116873,79803,-120754,-84790,0
C00696=40225,38253,-125973,74551,-121303,-87664,0
C00697=40226,38194,-125976,74566,-121328,-87635,0
C00698=36369,42537,-115581,79778,-121155,-84458,0
C00699=41037,38225,-125916,73749,-121788,-87735,0
C00700=40031,37676,-127220,74600,-120941,-87923,0
C00701=35405,42003,-116828,80533,-120312,-84657,0
C00702=36291,42493,-115684,79838,-121087,-84475,0
C00703=35675,42905,-114701,80556,-120866,-84142,0
C00704=36549,43410,-113524,79890,-121651,-83952,0
C00705=42267,38174,-126062,72472,-122424,-87953,0
C00706=39899,36880,-129135,74485,-120435,-88389,0
C00707=34302,42161,-116437,81632,-119674,-84421,0
C00708=35205,42644,-115311,80921,-120452,-84240,0
C00709=34969,42918,-114661,81229,-120412,-84043,0
C00710=35437,43179,-114052,80867,-120826,-83945,0
C00711=35621,42967,-114554,80627,-120857,-84097,0
C00712=36182,42604,-115419,79978,-121065,-84392,0
C00713=36146,41987,-116876,79817,-120774,-84763,0
C00714=40226,38194,-125976,74566,-121328,-87635,0
C00715=40226,38136,-125981,74581,-121354,-87606,0
C00716=36369,42484,-115584,79792,-121175,-84431,0
C00717=41038,38167,-125921,73765,-121815,-87707,0
C00718=40031,37617,-127223,74614,-120967,-87893,0
C00719=35405,41950,-116831,80546,-120332,-84629,0
C00720=36291,42440,-115688,79852,-121106,-84448,0
C00721=35675,42853,-114705,80570,-120885,-84115,0
C00722=36549,43358,-113528,79904,-121669,-83926,0
C00723=42268,38115,-126067,72488,-122452,-87924,0
C00724=39899,36820,-129140,74500,-120463,-88359,0
C00725=34303,42108,-116440,81645,-119693,-84394,0
C00726=35205,42591,-115315,80934,-120472,-84214,0
C00727=34969,42865,-114665,81242,-120430,-84016,0
C00728=35438,43127,-114056,80881,-120844,-83918,0
C00729=35621,42915,-114558,80641,-120876,-84071,0
C00730=36182,42552,-115422,79992,-121084,-84365,0
C00731=36146,41934,-116879,79831,-120795,-84736,0
C00732=40226,38136,-125981,74581,-121354,-87606,0
C00733=40227,38078,-125984,74597,-121381,-87577,0
C00734=36369,42432,-115589,79806,-121195,-84404,0
C00735=41038,38109,-125924,73780,-121842,-87678,0
C00736=40031,37558,-127228,74629,-120993,-87863,0
C00737=35406,41897,-116835,80560,-120351,-84602,0
C00738=36291,42387,-115692,79866,-121126,-84421,0
C00739=35675,42800,-114709,80583,-120904,-84088,0
C00740=36549,43307,-113532,79918,-121689,-83900,0
C00741=42268,38057,-126070,72504,-122479,-87895,0
C00742=39900,36759,-129143,74515,-120490,-88329,0
C00743=34303,42055,-116444,81658,-119711,-84367,0
C00744=35205,42538,-115319,80948,-120490,-84186,0
C00745=34969,42813,-114668,81255,-120449,-83989,0
C00746=35438,43075,-114060,80894,-120864,-83891,0
C00747=35621,42863,-114562,80654,-120895,-84044,0
C00748=36183,42499,-115426,80006,-121104,-84338,0
C00749=36147,41881,-116884,79845,-120814,-84708,0
C00750=40227,38078,-125984,74597,-121381,-87577,0
C00751=40227,38020,-125989,74612,-121407,-87548,0
C00752=36370,42379,-115592,79820,-121214,-84377,0
C00753=41039,38051,-125928,73796,-121869,-87649,0
C00754=40032,37499,-127231,74645,-121020,-87834,0
C00755=35406,41843,-116839,80573,-120371,-84574,0
C00756=36292,42335,-115696,79880,-121145,-84393,0
C00757=35676,42748,-114713,80597,-120923,-84061,0
C00758=36550,43255,-113536,79932,-121708,-83873,0
C00759=42269,37999,-126075,72519,-122508,-87866,0
C00760=39900,36699,-129148,74530,-120518,-88299,0
C00761=34303,42002,-116449,81671,-119729,-84339,0
C00762=35206,42486,-115322,80961,-120508,-84159,0
C00763=34970,42761,-114672,81269,-120467,-83962,0
C00764=35438,43023,-114064,80908,-120882,-83864,0
C00765=35621,42810,-114566,80668,-120913,-84017,0
C00766=36183,42447,-115430,80020,-121123,-84311,0
C00767=36147,41828,-116888,79859,-120834,-84681,0
C00768=40227,38020,-125989,74612,-121407,-87548,0
C00769=40227,37961,-125992,74627,-121434,-87519,0
C00770=36370,42326,-115596,79834,-121234,-84350,0
C00771=41039,37993,-125933,73811,-121896,-87620,0
C00772=40032,37440,-127236,74660,-121047,-87804,0
C00773=35406,41790,-116843,80587,-120389,-84547,0
C00774=36292,42282,-115699,79894,-121165,-84366,0
C00775=35676,42696,-114716,80611,-120942,-84034,0
C00776=36550,43203,-113539,79946,-121728,-83846,0
C00777=42269,37940,-126078,72535,-122536,-87837,0
C00778=39901,36639,-129151,74544,-120544,-88269,0
C00779=34303,41949,-116452,81684,-119748,-84312,0
C00780=35206,42434,-115326,80975,-120527,-84132,0
C00781=34970,42709,-114676,81282,-120486,-83935,0
C00782=35439,42971,-114067,80922,-120900,-83838,0
C00783=35622,42758,-114569,80682,-120933,-83990,0
C00784=36183,42394,-115434,80034,-121143,-84284,0
C00785=36147,41774,-116891,79873,-120854,-84653,0
C00786=40227,37961,-125992,74627,-121434,-87519,0
C00787=40228,37903,-125996,74642,-121460,-87490,0
C00788=36370,42274,-115599,79848,-121254,-84323,0
C00789=41039,37934,-125936,73827,-121923,-87590,0
C00790=40033,37381,-127239,74675,-121074,-87775,0
C00791=35407,41737,-116846,80600,-120409,-84519,0
C00792=36292,42229,-115703,79908,-121184,-84339,0
C00793=35676,42644,-114720,80625,-120960,-84008,0
C00794=36550,43152,-113543,79961,-121746,-83819,0
C00795=42270,37882,-126082,72551,-122564,-87809,0
C00796=39901,36579,-129155,74559,-120572,-88239,0
C00797=34304,41896,-116455,81697,-119766,-84284,0
C00798=35206,42381,-115329,80988,-120546,-84104,0
C00799=34970,42657,-114679,81296,-120504,-83908,0
C00800=35439,42919,-114071,80935,-120919,-83810,0
C00801=35622,42706,-114573,80696,-120951,-83963,0
C00802=36184,42342,-115437,80048,-121162,-84256,0
C00803=36148,41721,-116894,79887,-120874,-84626,0
C00804=40228,37903,-125996,74642,-121460,-87490,0
C00805=40228,37845,-125999,74658,-121486,-87460,0
C00806=36371,42221,-115603,79862,-121274,-84295,0
C00807=41040,37876,-125939,73842,-121950,-87561,0
C00808=40033,37322,-127243,74690,-121100,-87745,0
C00809=35407,41684,-116850,80614,-120428,-84492,0
C00810=36293,42177,-115706,79922,-121204,-84312,0
C00811=35677,42592,-114723,80639,-120980,-83980,0
C00812=36551,43100,-113546,79975,-121766,-83792,0
C00813=42270,37824,-126085,72567,-122592,-87780,0
C00814=39901,36519,-129158,74574,-120599,-88209,0
C00815=34304,41843,-116459,81710,-119785,-84256,0
C00816=35206,42329,-115333,81002,-120565,-84077,0
C00817=34971,42605,-114683,81309,-120522,-83881,0
C00818=35439,42867,-114074,80949,-120937,-83784,0
C00819=35623,42654,-114576,80709,-120969,-83936,0
C00820=36184,42289,-115441,80062,-121182,-84230,0
C00821=36148,41668,-116898,79901,-120893,-84598,0
C00822=40228,37845,-125999,74658,-121486,-87460,0
C00823=40229,37787,-126003,74673,-121513,-87431,0
C00824=36371,42169,-115606,79876,-121293,-84268,0
C00825=41040,37818,-125943,73858,-121977,-87532,0
C00826=40033,37263,-127246,74705,-121127,-87715,0
C00827=35407,41631,-116853,80628,-120448,-84464,0
C00828=36293,42124,-115710,79936,-121223,-84284,0
C00829=35677,42540,-114727,80652,-120998,-83953,0
C00830=36551,43048,-113550,79989,-121785,-83766,0
C00831=42270,37766,-126089,72584,-122621,-87751,0
C00832=39902,36458,-129163,74589,-120627,-88178,0
C00833=34305,41790,-116462,81723,-119803,-84229,0
C00834=35207,42276,-115336,81015,-120583,-84050,0
C00835=34971,42552,-114686,81323,-120541,-83854,0
C00836=35440,42815,-114078,80963,-120956,-83756,0
C00837=35623,42602,-114580,80723,-120989,-83908,0
C00838=36184,42237,-115444,80076,-121201,-84202,0
C00839=36148,41615,-116901,79915,-120913,-84571,0
C00840=40229,37787,-126003,74673,-121513,-87431,0
C00841=40229,37729,-126006,74688,-121538,-87402,0
C00842=36371,42116,-115610,79890,-121313,-84241,0
C00843=41041,37760,-125946,73874,-122004,-87503,0
C00844=40034,37204,-127249,74720,-121153,-87686,0
C00845=35408,41578,-116856,80641,-120467,-84436,0
C00846=36293,42072,-115713,79951,-121244,-84257,0
C00847=35677,42488,-114730,80666,-121018,-83926,0
C00848=36551,42997,-113553,80003,-121804,-83739,0
C00849=42271,37708,-126092,72600,-122648,-87722,0
C00850=39902,36398,-129166,74605,-120653,-88148,0
C00851=34305,41738,-116466,81736,-119821,-84201,0
C00852=35207,42224,-115340,81029,-120603,-84023,0
C00853=34971,42500,-114689,81336,-120559,-83826,0
C00854=35440,42764,-114081,80977,-120974,-83730,0
C00855=35623,42550,-114583,80737,-121007,-83882,0
C00856=36184,42184,-115448,80090,-121221,-84175,0
C00857=36149,41562,-116905,79929,-120934,-84543,0
C00858=40229,37729,-126006,74688,-121538,-87402,0
C00859=40229,37671,-126010,74704,-121565,-87372,0
C00860=36372,42064,-115613,79905,-121332,-84214,0
C00861=41041,37702,-125950,73890,-122031,-87474,0
C00862=40034,37145,-127253,74736,-121181,-87656,0
C00863=35408,41525,-116860,80655,-120486,-84409,0
C00864=36294,42019,-115717,79965,-121263,-84230,0
C00865=35678,42435,-114733,80680,-121036,-83899,0
C00866=36552,42945,-113556,80018,-121823,-83712,0
C00867=42271,37650,-126096,72616,-122677,-87693,0
C00868=39903,36338,-129170,74620,-120681,-88118,0
C00869=34305,41685,-116469,81750,-119840,-84174,0
C00870=35207,42172,-115343,81043,-120621,-83995,0
C00871=34972,42448,-114693,81350,-120577,-83799,0
C00872=35440,42712,-114084,80990,-120992,-83702,0
C00873=35623,42498,-114586,80751,-121027,-83854,0
C00874=36185,42132,-115450,80104,-121241,-84148,0
C00875=36149,41509,-116908,79943,-120953,-84516,0
C00876=40229,37671,-126010,74704,-121565,-87372,0
C00877=40230,37613,-126013,74719,-121591,-87343,0
C00878=36372,42011,-115615,79919,-121352,-84186,0
C00879=41041,37644,-125953,73905,-122058,-87444,0
C00880=40035,37087,-127256,74751,-121207,-87627,0
C00881=35408,41472,-116862,80669,-120505,-84381,0
C00882=36294,41967,-115719,79979,-121283,-84202,0
C00883=35678,42384,-114736,80694,-121055,-83872,0
C00884=36552,42894,-113559,80032,-121843,-83685,0
C00885=42272,37591,-126099,72632,-122705,-87664,0
C00886=39903,36278,-129172,74635,-120708,-88087,0
C00887=34305,41632,-116472,81763,-119858,-84146,0
C00888=35208,42119,-115346,81056,-120639,-83968,0
C00889=34972,42396,-114696,81363,-120596,-83773,0
C00890=35441,42660,-114087,81004,-121012,-83676,0
C00891=35624,42446,-114589,80765,-121045,-83827,0
C00892=36185,42080,-115453,80118,-121260,-84121,0
C00893=36149,41456,-116912,79957,-120973,-84488,0
C00894=40230,37613,-126013,74719,-121591,-87343,0
C00895=40230,37555,-126016,74735,-121617,-87314,0
C00896=36372,41959,-115619,79933,-121372,-84159,0
C00897=41042,37586,-125957,73921,-122085,-87415,0
C00898=40035,37028,-127260,74766,-121234,-87596,0
C00899=35409,41419,-116866,80683,-120525,-84354,0
C00900=36294,41914,-115722,79993,-121303,-84175,0
C00901=35678,42332,-114740,80708,-121074,-83844,0
C00902=36552,42843,-113562,80047,-121862,-83658,0
C00903=42272,37533,-126103,72648,-122733,-87635,0
C00904=39904,36218,-129175,74650,-120736,-88057,0
C00905=34306,41579,-116475,81776,-119876,-84118,0
C00906=35208,42067,-115349,81070,-120658,-83941,0
C00907=34972,42344,-114699,81377,-120614,-83745,0
C00908=35441,42609,-114090,81018,-121030,-83648,0
C00909=35624,42394,-114592,80779,-121064,-83800,0
C00910=36185,42027,-115457,80132,-121280,-84093,0
C00911=36150,41403,-116914,79971,-120993,-84461,0
C00912=40230,37555,-126016,74735,-121617,-87314,0
C00913=40231,37497,-126020,74750,-121644,-87284,0
C00914=36373,41907,-115622,79948,-121391,-84132,0
C00915=41042,37528,-125959,73937,-122112,-87386,0
C00916=40035,36969,-127262,74782,-121260,-87567,0
C00917=35409,41366,-116869,80696,-120544,-84326,0
C00918=36295,41862,-115726,80007,-121322,-84148,0
C00919=35679,42280,-114742,80722,-121093,-83817,0
C00920=36553,42791,-113565,80061,-121881,-83632,0
C00921=42273,37475,-126106,72665,-122761,-87605,0
C00922=39904,36158,-129179,74665,-120764,-88027,0
C00923=34306,41526,-116477,81789,-119895,-84091,0
C00924=35208,42015,-115352,81084,-120677,-83914,0
C00925=34973,42293,-114702,81391,-120633,-83718,0
C00926=35441,42557,-114093,81032,-121049,-83621,0
C00927=35624,42343,-114595,80793,-121083,-83773,0
C00928=36186,41975,-115459,80147,-121299,-84066,0
C00929=36150,41350,-116917,79985,-121013,-84433,0
C00930=40231,37497,-126020,74750,-121644,-87284,0
C00931=40231,37439,-126022,74766,-121670,-87255,0
C00932=36373,41854,-115625,79962,-121412,-84104,0
C00933=41043,37471,-125962,73953,-122139,-87357,0
C00934=40036,36910,-127266,74797,-121286,-87537,0
C00935=35409,41313,-116871,80710,-120564,-84298,0
C00936=36295,41810,-115728,80022,-121342,-84121,0
C00937=35679,42228,-114745,80736,-121112,-83790,0
C00938=36553,42740,-113568,80076,-121900,-83604,0
C00939=42273,37418,-126108,72681,-122790,-87576,0
C00940=39904,36098,-129182,74680,-120790,-87996,0
C00941=34306,41474,-116481,81803,-119913,-84063,0
C00942=35209,41963,-115355,81098,-120696,-83886,0
C00943=34973,42241,-114705,81404,-120651,-83691,0
C00944=35442,42505,-114096,81046,-121067,-83594,0
C00945=35625,42291,-114598,80807,-121101,-83746,0
C00946=36186,41923,-115463,80161,-121319,-84039,0
C00947=36150,41297,-116920,79999,-121033,-84405,0
C00948=40231,37439,-126022,74766,-121670,-87255,0
C00949=40231,37381,-126026,74781,-121697,-87225,0
C00950=36373,41802,-115628,79976,-121431,-84077,0
C00951=41043,37413,-125965,73969,-122166,-87327,0
C00952=40036,36852,-127269,74812,-121314,-87507,0
C00953=35410,41260,-116875,80724,-120582,-84270,0
C00954=36295,41757,-115731,80036,-121361,-84093,0
C00955=35679,42176,-114748,80750,-121130,-83763,0
C00956=36553,42689,-113571,80090,-121920,-83578,0
C00957=42273,37360,-126112,72697,-122817,-87547,0
C00958=39905,36038,-129185,74696,-120818,-87966,0
C00959=34307,41421,-116483,81816,-119932,-84035,0
C00960=35209,41911,-115358,81112,-120714,-83858,0
C00961=34973,42189,-114707,81418,-120669,-83663,0
C00962=35442,42454,-114099,81060,-121085,-83567,0
C00963=35625,42239,-114601,80821,-121121,-83719,0
C00964=36187,41871,-115465,80175,-121338,-84011,0
C00965=36151,41244,-116923,80013,-121053,-84377,0
C00966=40231,37381,-126026,74781,-121697,-87225,0
C00967=40232,37323,-126028,74797,-121723,-87196,0
C00968=36374,41750,-115630,79991,-121451,-84049,0
C00969=41043,37355,-125968,73985,-122193,-87298,0
C00970=40037,36793,-127271,74828,-121340,-87478,0
C00971=35410,41207,-116877,80738,-120602,-84243,0
C00972=36296,41705,-115734,80050,-121381,-84066,0
C00973=35680,42124,-114751,80764,-121150,-83735,0
C00974=36554,42637,-113573,80105,-121939,-83550,0
C00975=42274,37302,-126114,72714,-122846,-87518,0
C00976=39905,35978,-129188,74711,-120845,-87936,0
C00977=34307,41368,-116486,81829,-119950,-84008,0
C00978=35209,41859,-115360,81125,-120734,-83831,0
C00979=34974,42137,-114710,81432,-120688,-83636,0
C00980=35442,42402,-114101,81074,-121104,-83540,0
C00981=35625,42187,-114604,80835,-121139,-83691,0
C00982=36187,41819,-115468,80189,-121358,-83984,0
C00983=36151,41191,-116925,80028,-121073,-84350,0
C00984=40232,37323,-126028,74797,-121723,-87196,0
C00985=40232,37266,-126031,74813,-121750,-87166,0
C00986=36374,41698,-115633,80005,-121470,-84022,0
C00987=41044,37297,-125970,74001,-122220,-87269,0
C00988=40037,36735,-127274,74843,-121367,-87447,0
C00989=35410,41154,-116879,80752,-120621,-84215,0
C00990=36296,41653,-115736,80065,-121400,-84038,0
C00991=35680,42072,-114753,80779,-121168,-83708,0
C00992=36554,42586,-113576,80119,-121958,-83524,0
C00993=42274,37244,-126118,72730,-122873,-87489,0
C00994=39906,35919,-129190,74726,-120873,-87905,0
C00995=34307,41316,-116489,81843,-119968,-83980,0
C00996=35210,41806,-115363,81139,-120752,-83804,0
C00997=34974,42085,-114713,81446,-120706,-83608,0
C00998=35443,42351,-114104,81088,-121123,-83513,0
C00999=35626,42135,-114606,80849,-121158,-83664,0
C01000=36187,41767,-115471,80204,-121377,-83956,0
C01001=36151,41138,-116929,80042,-121092,-84322,0
C01002=40232,37266,-126031,74813,-121750,-87166,0
C01003=40233,37208,-126034,74828,-121776,-87137,0
C01004=36374,41646,-115635,80019,-121490,-83995,0
C01005=41044,37240,-125974,74017,-122247,-87239,0
C01006=40037,36676,-127277,74859,-121393,-87418,0
C01007=35411,41102,-116882,80766,-120641,-84187,0
C01008=36296,41601,-115738,80079,-121421,-84010,0
C01009=35680,42021,-114756,80793,-121188,-83681,0
C01010=36554,42535,-113579,80134,-121977,-83496,0
C01011=42275,37186,-126120,72747,-122902,-87460,0
C01012=39906,35859,-129194,74742,-120900,-87875,0
C01013=34308,41263,-116491,81856,-119987,-83952,0
C01014=35210,41754,-115366,81153,-120771,-83776,0
C01015=34974,42034,-114715,81459,-120725,-83581,0
C01016=35443,42299,-114107,81102,-121142,-83485,0
C01017=35626,42084,-114609,80863,-121177,-83637,0
C01018=36188,41714,-115473,80218,-121397,-83929,0
C01019=36152,41086,-116931,80056,-121113,-84294,0
C01020=40233,37208,-126034,74828,-121776,-87137,0
C01021=40233,37150,-126036,74844,-121802,-87107,0
C01022=36375,41593,-115638,80034,-121509,-83967,0
C01023=41045,37182,-125976,74033,-122275,-87210,0
C01024=40038,36618,-127279,74875,-121421,-87388,0
C01025=35411,41049,-116885,80780,-120660,-84159,0
C01026=36297,41548,-115742,80094,-121440,-83983,0
C01027=35681,41969,-114758,80807,-121206,-83654,0
C01028=36555,42484,-113581,80148,-121997,-83469,0
C01029=42275,37128,-126122,72763,-122930,-87430,0
C01030=39907,35799,-129196,74757,-120928,-87844,0
C01031=34308,41211,-116493,81870,-120005,-83924,0
C01032=35210,41702,-115368,81167,-120790,-83749,0
C01033=34975,41982,-114718,81473,-120743,-83554,0
C01034=35443,42248,-114109,81116,-121160,-83458,0
C01035=35626,42032,-114611,80877,-121196,-83609,0
C01036=36188,41662,-115475,80233,-121416,-83901,0
C01037=36152,41033,-116933,80071,-121132,-84266,0
C01038=40233,37150,-126036,74844,-121802,-87107,0
C01039=40233,37092,-126038,74860,-121829,-87078,0
C01040=36375,41541,-115641,80048,-121529,-83940,0
C01041=41045,37124,-125978,74049,-122301,-87180,0
C01042=40038,36559,-127282,74890,-121447,-87358,0
C01043=35411,40996,-116888,80794,-120679,-84131,0
C01044=36297,41496,-115744,80108,-121460,-83955,0
C01045=35681,41917,-114761,80821,-121226,-83626,0
C01046=36555,42432,-113583,80163,-122016,-83442,0
C01047=42276,37071,-126124,72780,-122958,-87401,0
C01048=39907,35739,-129198,74773,-120954,-87813,0
C01049=34308,41158,-116497,81883,-120022,-83896,0
C01050=35211,41650,-115371,81181,-120808,-83721,0
C01051=34975,41930,-114720,81487,-120761,-83526,0
C01052=35444,42197,-114111,81130,-121178,-83431,0
C01053=35627,41981,-114614,80891,-121215,-83582,0
C01054=36188,41610,-115477,80247,-121436,-83874,0
C01055=36152,40980,-116936,80085,-121152,-84238,0
C01056=40233,37092,-126038,74860,-121829,-87078,0
C01057=40234,37035,-126041,74876,-121855,-87048,0
C01058=36375,41489,-115643,80063,-121550,-83912,0
C01059=41046,37067,-125981,74065,-122329,-87151,0
C01060=40039,36501,-127284,74906,-121474,-87328,0
C01061=35412,40944,-116890,80808,-120698,-84103,0
C01062=36297,41444,-115746,80123,-121480,-83928,0
C01063=35681,41866,-114763,80835,-121244,-83598,0
C01064=36555,42381,-113586,80178,-122035,-83415,0
C01065=42276,37013,-126127,72796,-122986,-87371,0
C01066=39907,35680,-129201,74788,-120982,-87783,0
C01067=34309,41106,-116499,81897,-120041,-83868,0
C01068=35211,41599,-115373,81195,-120827,-83694,0
C01069=34975,41879,-114722,81501,-120780,-83499,0
C01070=35444,42145,-114114,81144,-121197,-83403,0
C01071=35627,41929,-114616,80906,-121234,-83554,0
C01072=36189,41558,-115480,80261,-121455,-83846,0
C01073=36153,40927,-116938,80099,-121173,-84211,0
C01074=40234,37035,-126041,74876,-121855,-87048,0
C01075=40234,36977,-126044,74892,-121882,-87019,0
C01076=36376,41437,-115645,80078,-121569,-83885,0
C01077=41046,37009,-125983,74081,-122355,-87121,0
C01078=40039,36442,-127286,74922,-121501,-87298,0
C01079=35412,40891,-116892,80822,-120718,-84075,0
C01080=36298,41392,-115749,80137,-121499,-83900,0
C01081=35682,41814,-114765,80849,-121263,-83571,0
C01082=36556,42330,-113588,80192,-122054,-83388,0
C01083=42276,36955,-126129,72813,-123015,-87342,0
C01084=39908,35620,-129203,74804,-121010,-87753,0
C01085=34309,41053,-116501,81910,-120060,-83840,0
C01086=35211,41547,-115375,81209,-120846,-83666,0
C01087=34976,41827,-114725,81515,-120798,-83471,0
C01088=35444,42094,-114116,81158,-121215,-83376,0
C01089=35627,41877,-114618,80920,-121252,-83527,0
C01090=36189,41506,-115482,80276,-121475,-83819,0
C01091=36153,40875,-116940,80114,-121192,-84183,0
C01092=40234,36977,-126044,74892,-121882,-87019,0
C01093=40235,36920,-126045,74907,-121908,-86988,0
C01094=36376,41385,-115646,80092,-121589,-83857,0
C01095=41046,36951,-125985,74097,-122383,-87092,0
C01096=40040,36384,-127289,74937,-121528,-87267,0
C01097=35412,40838,-116893,80836,-120737,-84048,0
C01098=36298,41340,-115750,80152,-121519,-83873,0
C01099=35682,41762,-114767,80864,-121282,-83544,0
C01100=36556,42279,-113590,80207,-122074,-83361,0
C01101=42277,36898,-126131,72830,-123042,-87313,0
C01102=39908,35560,-129205,74820,-121037,-87722,0
C01103=34309,41001,-116503,81924,-120079,-83813,0
C01104=35212,41495,-115378,81223,-120865,-83638,0
C01105=34976,41775,-114727,81529,-120816,-83444,0
C01106=35445,42043,-114118,81173,-121235,-83349,0
C01107=35628,41826,-114620,80934,-121272,-83500,0
C01108=36189,41454,-115484,80290,-121494,-83791,0
C01109=36153,40822,-116943,80128,-121212,-84155,0
C01110=40235,36920,-126045,74907,-121908,-86988,0
C01111=40235,36862,-126047,74923,-121935,-86959,0
C01112=36376,41333,-115649,80107,-121608,-83829,0
C01113=41047,36894,-125988,74114,-122410,-87062,0
C01114=40040,36326,-127291,74953,-121554,-87237,0
C01115=35413,40786,-116896,80850,-120757,-84020,0
C01116=36298,41288,-115752,80166,-121538,-83845,0
C01117=35682,41711,-114769,80878,-121301,-83516,0
C01118=36556,42228,-113592,80222,-122093,-83333,0
C01119=42277,36840,-126134,72846,-123071,-87283,0
C01120=39909,35501,-129208,74835,-121065,-87691,0
C01121=34310,40949,-116505,81937,-120097,-83785,0
C01122=35212,41443,-115379,81237,-120883,-83611,0
C01123=34976,41724,-114729,81543,-120835,-83416,0
C01124=35445,41991,-114120,81187,-121253,-83322,0
C01125=35628,41774,-114622,80948,-121290,-83472,0
C01126=36189,41403,-115487,80305,-121514,-83764,0
C01127=36154,40770,-116945,80143,-121232,-84127,0
C01128=40235,36862,-126047,74923,-121935,-86959,0
C01129=40236,36805,-126050,74939,-121961,-86929,0
C01130=36377,41281,-115651,80121,-121628,-83802,0
C01131=41047,36836,-125990,74130,-122437,-87032,0
C01132=40040,36267,-127293,74969,-121581,-87208,0
C01133=35413,40733,-116898,80864,-120776,-83991,0
C01134=36299,41236,-115754,80181,-121559,-83817,0
C01135=35683,41659,-114771,80892,-121320,-83489,0
C01136=36557,42177,-113594,80237,-122113,-83307,0
C01137=42278,36782,-126136,72863,-123100,-87254,0
C01138=39909,35441,-129210,74851,-121092,-87660,0
C01139=34310,40896,-116507,81951,-120115,-83756,0
C01140=35212,41391,-115381,81251,-120903,-83583,0
C01141=34976,41672,-114731,81557,-120853,-83389,0
C01142=35445,41940,-114122,81201,-121272,-83294,0
C01143=35628,41723,-114624,80963,-121309,-83445,0
C01144=36190,41351,-115489,80320,-121534,-83736,0
C01145=36154,40717,-116946,80157,-121252,-84099,0
C01146=40236,36805,-126050,74939,-121961,-86929,0
C01147=40236,36747,-126052,74955,-121987,-86900,0
C01148=36377,41230,-115653,80136,-121648,-83774,0
C01149=41048,36779,-125991,74146,-122464,-87003,0
C01150=40041,36209,-127295,74985,-121608,-87178,0
C01151=35413,40681,-116900,80878,-120795,-83963,0
C01152=36299,41184,-115757,80196,-121578,-83789,0
C01153=35683,41608,-114773,80907,-121339,-83461,0
C01154=36557,42126,-113596,80252,-122131,-83279,0
C01155=42278,36725,-126138,72880,-123127,-87224,0
C01156=39909,35382,-129212,74867,-121120,-87630,0
C01157=34310,40844,-116509,81964,-120134,-83728,0
C01158=35213,41339,-115383,81265,-120921,-83555,0
C01159=34977,41621,-114733,81571,-120872,-83361,0
C01160=35446,41889,-114124,81215,-121290,-83267,0
//INST
///DATE 2025/02/20 16:20
///COMM Generated using RoboDK
///ATTR SC,RW
///GROUP1 RB1
NOP
MOVL C00000 V=60.0 PL=1
MOVL C00001 V=130.0 PL=1
MOVL C00002 V=30.0 PL=1
MOVL C00003 V=30.0 PL=1
MOVL C00004 V=30.0 PL=1
MOVL C00005 V=30.0 PL=1
MOVL C00006 V=30.0 PL=1
MOVL C00007 V=30.0 PL=1
MOVL C00008 V=30.0 PL=1
MOVL C00009 V=30.0 PL=1
MOVL C00010 V=130.0 PL=1
MOVL C00011 V=130.0 PL=1
MOVL C00012 V=20.0 PL=1
MOVL C00013 V=130.0 PL=1
MOVL C00014 V=130.0 PL=1
MOVL C00015 V=60.0 PL=1
MOVL C00016 V=60.0 PL=1
MOVL C00017 V=60.0 PL=1
MOVL C00018 V=60.0 PL=1
MOVL C00019 V=130.0 PL=1
MOVL C00020 V=30.0 PL=1
MOVL C00021 V=30.0 PL=1
MOVL C00022 V=30.0 PL=1
MOVL C00023 V=30.0 PL=1
MOVL C00024 V=30.0 PL=1
MOVL C00025 V=30.0 PL=1
MOVL C00026 V=30.0 PL=1
MOVL C00027 V=30.0 PL=1
MOVL C00028 V=130.0 PL=1
MOVL C00029 V=130.0 PL=1
MOVL C00030 V=20.0 PL=1
MOVL C00031 V=130.0 PL=1
MOVL C00032 V=130.0 PL=1
MOVL C00033 V=60.0 PL=1
MOVL C00034 V=60.0 PL=1
MOVL C00035 V=60.0 PL=1
MOVL C00036 V=60.0 PL=1
MOVL C00037 V=130.0 PL=1
MOVL C00038 V=30.0 PL=1
MOVL C00039 V=30.0 PL=1
MOVL C00040 V=30.0 PL=1
MOVL C00041 V=30.0 PL=1
MOVL C00042 V=30.0 PL=1
MOVL C00043 V=30.0 PL=1
MOVL C00044 V=30.0 PL=1
MOVL C00045 V=30.0 PL=1
MOVL C00046 V=130.0 PL=1
MOVL C00047 V=130.0 PL=1
MOVL C00048 V=20.0 PL=1
MOVL C00049 V=130.0 PL=1
MOVL C00050 V=130.0 PL=1
MOVL C00051 V=60.0 PL=1
MOVL C00052 V=60.0 PL=1
MOVL C00053 V=60.0 PL=1
MOVL C00054 V=60.0 PL=1
MOVL C00055 V=130.0 PL=1
MOVL C00056 V=30.0 PL=1
MOVL C00057 V=30.0 PL=1
MOVL C00058 V=30.0 PL=1
MOVL C00059 V=30.0 PL=1
MOVL C00060 V=30.0 PL=1
MOVL C00061 V=30.0 PL=1
MOVL C00062 V=30.0 PL=1
MOVL C00063 V=30.0 PL=1
MOVL C00064 V=130.0 PL=1
MOVL C00065 V=130.0 PL=1
MOVL C00066 V=20.0 PL=1
MOVL C00067 V=130.0 PL=1
MOVL C00068 V=130.0 PL=1
MOVL C00069 V=60.0 PL=1
MOVL C00070 V=60.0 PL=1
MOVL C00071 V=60.0 PL=1
MOVL C00072 V=60.0 PL=1
MOVL C00073 V=130.0 PL=1
MOVL C00074 V=30.0 PL=1
MOVL C00075 V=30.0 PL=1
MOVL C00076 V=30.0 PL=1
MOVL C00077 V=30.0 PL=1
MOVL C00078 V=30.0 PL=1
MOVL C00079 V=30.0 PL=1
MOVL C00080 V=30.0 PL=1
MOVL C00081 V=30.0 PL=1
MOVL C00082 V=130.0 PL=1
MOVL C00083 V=130.0 PL=1
MOVL C00084 V=20.0 PL=1
MOVL C00085 V=130.0 PL=1
MOVL C00086 V=130.0 PL=1
MOVL C00087 V=60.0 PL=1
MOVL C00088 V=60.0 PL=1
MOVL C00089 V=60.0 PL=1
MOVL C00090 V=60.0 PL=1
MOVL C00091 V=130.0 PL=1
MOVL C00092 V=30.0 PL=1
MOVL C00093 V=30.0 PL=1
MOVL C00094 V=30.0 PL=1
MOVL C00095 V=30.0 PL=1
MOVL C00096 V=30.0 PL=1
MOVL C00097 V=30.0 PL=1
MOVL C00098 V=30.0 PL=1
MOVL C00099 V=30.0 PL=1
MOVL C00100 V=130.0 PL=1
MOVL C00101 V=130.0 PL=1
MOVL C00102 V=20.0 PL=1
MOVL C00103 V=130.0 PL=1
MOVL C00104 V=130.0 PL=1
MOVL C00105 V=60.0 PL=1
MOVL C00106 V=60.0 PL=1
MOVL C00107 V=60.0 PL=1
MOVL C00108 V=60.0 PL=1
MOVL C00109 V=130.0 PL=1
MOVL C00110 V=30.0 PL=1
MOVL C00111 V=30.0 PL=1
MOVL C00112 V=30.0 PL=1
MOVL C00113 V=30.0 PL=1
MOVL C00114 V=30.0 PL=1
MOVL C00115 V=30.0 PL=1
MOVL C00116 V=30.0 PL=1
MOVL C00117 V=30.0 PL=1
MOVL C00118 V=130.0 PL=1
MOVL C00119 V=130.0 PL=1
MOVL C00120 V=20.0 PL=1
MOVL C00121 V=130.0 PL=1
MOVL C00122 V=130.0 PL=1
MOVL C00123 V=60.0 PL=1
MOVL C00124 V=60.0 PL=1
MOVL C00125 V=60.0 PL=1
MOVL C00126 V=60.0 PL=1
MOVL C00127 V=130.0 PL=1
MOVL C00128 V=30.0 PL=1
MOVL C00129 V=30.0 PL=1
MOVL C00130 V=30.0 PL=1
MOVL C00131 V=30.0 PL=1
MOVL C00132 V=30.0 PL=1
MOVL C00133 V=30.0 PL=1
MOVL C00134 V=30.0 PL=1
MOVL C00135 V=30.0 PL=1
MOVL C00136 V=130.0 PL=1
MOVL C00137 V=130.0 PL=1
MOVL C00138 V=20.0 PL=1
MOVL C00139 V=130.0 PL=1
MOVL C00140 V=130.0 PL=1
MOVL C00141 V=60.0 PL=1
MOVL C00142 V=60.0 PL=1
MOVL C00143 V=60.0 PL=1
MOVL C00144 V=60.0 PL=1
MOVL C00145 V=130.0 PL=1
MOVL C00146 V=30.0 PL=1
MOVL C00147 V=30.0 PL=1
MOVL C00148 V=30.0 PL=1
MOVL C00149 V=30.0 PL=1
MOVL C00150 V=30.0 PL=1
MOVL C00151 V=30.0 PL=1
MOVL C00152 V=30.0 PL=1
MOVL C00153 V=30.0 PL=1
MOVL C00154 V=130.0 PL=1
MOVL C00155 V=130.0 PL=1
MOVL C00156 V=20.0 PL=1
MOVL C00157 V=130.0 PL=1
MOVL C00158 V=130.0 PL=1
MOVL C00159 V=60.0 PL=1
MOVL C00160 V=60.0 PL=1
MOVL C00161 V=60.0 PL=1
MOVL C00162 V=60.0 PL=1
MOVL C00163 V=130.0 PL=1
MOVL C00164 V=30.0 PL=1
MOVL C00165 V=30.0 PL=1
MOVL C00166 V=30.0 PL=1
MOVL C00167 V=30.0 PL=1
MOVL C00168 V=30.0 PL=1
MOVL C00169 V=30.0 PL=1
MOVL C00170 V=30.0 PL=1
MOVL C00171 V=30.0 PL=1
MOVL C00172 V=130.0 PL=1
MOVL C00173 V=130.0 PL=1
MOVL C00174 V=20.0 PL=1
MOVL C00175 V=130.0 PL=1
MOVL C00176 V=130.0 PL=1
MOVL C00177 V=60.0 PL=1
MOVL C00178 V=60.0 PL=1
MOVL C00179 V=60.0 PL=1
MOVL C00180 V=60.0 PL=1
MOVL C00181 V=130.0 PL=1
MOVL C00182 V=30.0 PL=1
MOVL C00183 V=30.0 PL=1
MOVL C00184 V=30.0 PL=1
MOVL C00185 V=30.0 PL=1
MOVL C00186 V=30.0 PL=1
MOVL C00187 V=30.0 PL=1
MOVL C00188 V=30.0 PL=1
MOVL C00189 V=30.0 PL=1
MOVL C00190 V=130.0 PL=1
MOVL C00191 V=130.0 PL=1
MOVL C00192 V=20.0 PL=1
MOVL C00193 V=130.0 PL=1
MOVL C00194 V=130.0 PL=1
MOVL C00195 V=60.0 PL=1
MOVL C00196 V=60.0 PL=1
MOVL C00197 V=60.0 PL=1
MOVL C00198 V=60.0 PL=1
MOVL C00199 V=130.0 PL=1
MOVL C00200 V=30.0 PL=1
MOVL C00201 V=30.0 PL=1
MOVL C00202 V=30.0 PL=1
MOVL C00203 V=30.0 PL=1
MOVL C00204 V=30.0 PL=1
MOVL C00205 V=30.0 PL=1
MOVL C00206 V=30.0 PL=1
MOVL C00207 V=30.0 PL=1
MOVL C00208 V=130.0 PL=1
MOVL C00209 V=130.0 PL=1
MOVL C00210 V=20.0 PL=1
MOVL C00211 V=130.0 PL=1
MOVL C00212 V=130.0 PL=1
MOVL C00213 V=60.0 PL=1
MOVL C00214 V=60.0 PL=1
MOVL C00215 V=60.0 PL=1
MOVL C00216 V=60.0 PL=1
MOVL C00217 V=130.0 PL=1
MOVL C00218 V=30.0 PL=1
MOVL C00219 V=30.0 PL=1
MOVL C00220 V=30.0 PL=1
MOVL C00221 V=30.0 PL=1
MOVL C00222 V=30.0 PL=1
MOVL C00223 V=30.0 PL=1
MOVL C00224 V=30.0 PL=1
MOVL C00225 V=30.0 PL=1
MOVL C00226 V=130.0 PL=1
MOVL C00227 V=130.0 PL=1
MOVL C00228 V=20.0 PL=1
MOVL C00229 V=130.0 PL=1
MOVL C00230 V=130.0 PL=1
MOVL C00231 V=60.0 PL=1
MOVL C00232 V=60.0 PL=1
MOVL C00233 V=60.0 PL=1
MOVL C00234 V=60.0 PL=1
MOVL C00235 V=130.0 PL=1
MOVL C00236 V=30.0 PL=1
MOVL C00237 V=30.0 PL=1
MOVL C00238 V=30.0 PL=1
MOVL C00239 V=30.0 PL=1
MOVL C00240 V=30.0 PL=1
MOVL C00241 V=30.0 PL=1
MOVL C00242 V=30.0 PL=1
MOVL C00243 V=30.0 PL=1
MOVL C00244 V=130.0 PL=1
MOVL C00245 V=130.0 PL=1
MOVL C00246 V=20.0 PL=1
MOVL C00247 V=130.0 PL=1
MOVL C00248 V=130.0 PL=1
MOVL C00249 V=60.0 PL=1
MOVL C00250 V=60.0 PL=1
MOVL C00251 V=60.0 PL=1
MOVL C00252 V=60.0 PL=1
MOVL C00253 V=130.0 PL=1
MOVL C00254 V=30.0 PL=1
MOVL C00255 V=30.0 PL=1
MOVL C00256 V=30.0 PL=1
MOVL C00257 V=30.0 PL=1
MOVL C00258 V=30.0 PL=1
MOVL C00259 V=30.0 PL=1
MOVL C00260 V=30.0 PL=1
MOVL C00261 V=30.0 PL=1
MOVL C00262 V=130.0 PL=1
MOVL C00263 V=130.0 PL=1
MOVL C00264 V=20.0 PL=1
MOVL C00265 V=130.0 PL=1
MOVL C00266 V=130.0 PL=1
MOVL C00267 V=60.0 PL=1
MOVL C00268 V=60.0 PL=1
MOVL C00269 V=60.0 PL=1
MOVL C00270 V=60.0 PL=1
MOVL C00271 V=130.0 PL=1
MOVL C00272 V=30.0 PL=1
MOVL C00273 V=30.0 PL=1
MOVL C00274 V=30.0 PL=1
MOVL C00275 V=30.0 PL=1
MOVL C00276 V=30.0 PL=1
MOVL C00277 V=30.0 PL=1
MOVL C00278 V=30.0 PL=1
MOVL C00279 V=30.0 PL=1
MOVL C00280 V=130.0 PL=1
MOVL C00281 V=130.0 PL=1
MOVL C00282 V=20.0 PL=1
MOVL C00283 V=130.0 PL=1
MOVL C00284 V=130.0 PL=1
MOVL C00285 V=60.0 PL=1
MOVL C00286 V=60.0 PL=1
MOVL C00287 V=60.0 PL=1
MOVL C00288 V=60.0 PL=1
MOVL C00289 V=130.0 PL=1
MOVL C00290 V=30.0 PL=1
MOVL C00291 V=30.0 PL=1
MOVL C00292 V=30.0 PL=1
MOVL C00293 V=30.0 PL=1
MOVL C00294 V=30.0 PL=1
MOVL C00295 V=30.0 PL=1
MOVL C00296 V=30.0 PL=1
MOVL C00297 V=30.0 PL=1
MOVL C00298 V=130.0 PL=1
MOVL C00299 V=130.0 PL=1
MOVL C00300 V=20.0 PL=1
MOVL C00301 V=130.0 PL=1
MOVL C00302 V=130.0 PL=1
MOVL C00303 V=60.0 PL=1
MOVL C00304 V=60.0 PL=1
MOVL C00305 V=60.0 PL=1
MOVL C00306 V=60.0 PL=1
MOVL C00307 V=130.0 PL=1
MOVL C00308 V=30.0 PL=1
MOVL C00309 V=30.0 PL=1
MOVL C00310 V=30.0 PL=1
MOVL C00311 V=30.0 PL=1
MOVL C00312 V=30.0 PL=1
MOVL C00313 V=30.0 PL=1
MOVL C00314 V=30.0 PL=1
MOVL C00315 V=30.0 PL=1
MOVL C00316 V=130.0 PL=1
MOVL C00317 V=130.0 PL=1
MOVL C00318 V=20.0 PL=1
MOVL C00319 V=130.0 PL=1
MOVL C00320 V=130.0 PL=1
MOVL C00321 V=60.0 PL=1
MOVL C00322 V=60.0 PL=1
MOVL C00323 V=60.0 PL=1
MOVL C00324 V=60.0 PL=1
MOVL C00325 V=130.0 PL=1
MOVL C00326 V=30.0 PL=1
MOVL C00327 V=30.0 PL=1
MOVL C00328 V=30.0 PL=1
MOVL C00329 V=30.0 PL=1
MOVL C00330 V=30.0 PL=1
MOVL C00331 V=30.0 PL=1
MOVL C00332 V=30.0 PL=1
MOVL C00333 V=30.0 PL=1
MOVL C00334 V=130.0 PL=1
MOVL C00335 V=130.0 PL=1
MOVL C00336 V=20.0 PL=1
MOVL C00337 V=130.0 PL=1
MOVL C00338 V=130.0 PL=1
MOVL C00339 V=60.0 PL=1
MOVL C00340 V=60.0 PL=1
MOVL C00341 V=60.0 PL=1
MOVL C00342 V=60.0 PL=1
MOVL C00343 V=130.0 PL=1
MOVL C00344 V=30.0 PL=1
MOVL C00345 V=30.0 PL=1
MOVL C00346 V=30.0 PL=1
MOVL C00347 V=30.0 PL=1
MOVL C00348 V=30.0 PL=1
MOVL C00349 V=30.0 PL=1
MOVL C00350 V=30.0 PL=1
MOVL C00351 V=30.0 PL=1
MOVL C00352 V=130.0 PL=1
MOVL C00353 V=130.0 PL=1
MOVL C00354 V=20.0 PL=1
MOVL C00355 V=130.0 PL=1
MOVL C00356 V=130.0 PL=1
MOVL C00357 V=60.0 PL=1
MOVL C00358 V=60.0 PL=1
MOVL C00359 V=60.0 PL=1
MOVL C00360 V=60.0 PL=1
MOVL C00361 V=130.0 PL=1
MOVL C00362 V=30.0 PL=1
MOVL C00363 V=30.0 PL=1
MOVL C00364 V=30.0 PL=1
MOVL C00365 V=30.0 PL=1
MOVL C00366 V=30.0 PL=1
MOVL C00367 V=30.0 PL=1
MOVL C00368 V=30.0 PL=1
MOVL C00369 V=30.0 PL=1
MOVL C00370 V=130.0 PL=1
MOVL C00371 V=130.0 PL=1
MOVL C00372 V=20.0 PL=1
MOVL C00373 V=130.0 PL=1
MOVL C00374 V=130.0 PL=1
MOVL C00375 V=60.0 PL=1
MOVL C00376 V=60.0 PL=1
MOVL C00377 V=60.0 PL=1
MOVL C00378 V=60.0 PL=1
MOVL C00379 V=130.0 PL=1
MOVL C00380 V=30.0 PL=1
MOVL C00381 V=30.0 PL=1
MOVL C00382 V=30.0 PL=1
MOVL C00383 V=30.0 PL=1
MOVL C00384 V=30.0 PL=1
MOVL C00385 V=30.0 PL=1
MOVL C00386 V=30.0 PL=1
MOVL C00387 V=30.0 PL=1
MOVL C00388 V=130.0 PL=1
MOVL C00389 V=130.0 PL=1
MOVL C00390 V=20.0 PL=1
MOVL C00391 V=130.0 PL=1
MOVL C00392 V=130.0 PL=1
MOVL C00393 V=60.0 PL=1
MOVL C00394 V=60.0 PL=1
MOVL C00395 V=60.0 PL=1
MOVL C00396 V=60.0 PL=1
MOVL C00397 V=130.0 PL=1
MOVL C00398 V=30.0 PL=1
MOVL C00399 V=30.0 PL=1
MOVL C00400 V=30.0 PL=1
MOVL C00401 V=30.0 PL=1
MOVL C00402 V=30.0 PL=1
MOVL C00403 V=30.0 PL=1
MOVL C00404 V=30.0 PL=1
MOVL C00405 V=30.0 PL=1
MOVL C00406 V=130.0 PL=1
MOVL C00407 V=130.0 PL=1
MOVL C00408 V=20.0 PL=1
MOVL C00409 V=130.0 PL=1
MOVL C00410 V=130.0 PL=1
MOVL C00411 V=60.0 PL=1
MOVL C00412 V=60.0 PL=1
MOVL C00413 V=60.0 PL=1
MOVL C00414 V=60.0 PL=1
MOVL C00415 V=130.0 PL=1
MOVL C00416 V=30.0 PL=1
MOVL C00417 V=30.0 PL=1
MOVL C00418 V=30.0 PL=1
MOVL C00419 V=30.0 PL=1
MOVL C00420 V=30.0 PL=1
MOVL C00421 V=30.0 PL=1
MOVL C00422 V=30.0 PL=1
MOVL C00423 V=30.0 PL=1
MOVL C00424 V=130.0 PL=1
MOVL C00425 V=130.0 PL=1
MOVL C00426 V=20.0 PL=1
MOVL C00427 V=130.0 PL=1
MOVL C00428 V=130.0 PL=1
MOVL C00429 V=60.0 PL=1
MOVL C00430 V=60.0 PL=1
MOVL C00431 V=60.0 PL=1
MOVL C00432 V=60.0 PL=1
MOVL C00433 V=130.0 PL=1
MOVL C00434 V=30.0 PL=1
MOVL C00435 V=30.0 PL=1
MOVL C00436 V=30.0 PL=1
MOVL C00437 V=30.0 PL=1
MOVL C00438 V=30.0 PL=1
MOVL C00439 V=30.0 PL=1
MOVL C00440 V=30.0 PL=1
MOVL C00441 V=30.0 PL=1
MOVL C00442 V=130.0 PL=1
MOVL C00443 V=130.0 PL=1
MOVL C00444 V=20.0 PL=1
MOVL C00445 V=130.0 PL=1
MOVL C00446 V=130.0 PL=1
MOVL C00447 V=60.0 PL=1
MOVL C00448 V=60.0 PL=1
MOVL C00449 V=60.0 PL=1
MOVL C00450 V=60.0 PL=1
MOVL C00451 V=130.0 PL=1
MOVL C00452 V=30.0 PL=1
MOVL C00453 V=30.0 PL=1
MOVL C00454 V=30.0 PL=1
MOVL C00455 V=30.0 PL=1
MOVL C00456 V=30.0 PL=1
MOVL C00457 V=30.0 PL=1
MOVL C00458 V=30.0 PL=1
MOVL C00459 V=30.0 PL=1
MOVL C00460 V=130.0 PL=1
MOVL C00461 V=130.0 PL=1
MOVL C00462 V=20.0 PL=1
MOVL C00463 V=130.0 PL=1
MOVL C00464 V=130.0 PL=1
MOVL C00465 V=60.0 PL=1
MOVL C00466 V=60.0 PL=1
MOVL C00467 V=60.0 PL=1
MOVL C00468 V=60.0 PL=1
MOVL C00469 V=130.0 PL=1
MOVL C00470 V=30.0 PL=1
MOVL C00471 V=30.0 PL=1
MOVL C00472 V=30.0 PL=1
MOVL C00473 V=30.0 PL=1
MOVL C00474 V=30.0 PL=1
MOVL C00475 V=30.0 PL=1
MOVL C00476 V=30.0 PL=1
MOVL C00477 V=30.0 PL=1
MOVL C00478 V=130.0 PL=1
MOVL C00479 V=130.0 PL=1
MOVL C00480 V=20.0 PL=1
MOVL C00481 V=130.0 PL=1
MOVL C00482 V=130.0 PL=1
MOVL C00483 V=60.0 PL=1
MOVL C00484 V=60.0 PL=1
MOVL C00485 V=60.0 PL=1
MOVL C00486 V=60.0 PL=1
MOVL C00487 V=130.0 PL=1
MOVL C00488 V=30.0 PL=1
MOVL C00489 V=30.0 PL=1
MOVL C00490 V=30.0 PL=1
MOVL C00491 V=30.0 PL=1
MOVL C00492 V=30.0 PL=1
MOVL C00493 V=30.0 PL=1
MOVL C00494 V=30.0 PL=1
MOVL C00495 V=30.0 PL=1
MOVL C00496 V=130.0 PL=1
MOVL C00497 V=130.0 PL=1
MOVL C00498 V=20.0 PL=1
MOVL C00499 V=130.0 PL=1
MOVL C00500 V=130.0 PL=1
MOVL C00501 V=60.0 PL=1
MOVL C00502 V=60.0 PL=1
MOVL C00503 V=60.0 PL=1
MOVL C00504 V=60.0 PL=1
MOVL C00505 V=130.0 PL=1
MOVL C00506 V=30.0 PL=1
MOVL C00507 V=30.0 PL=1
MOVL C00508 V=30.0 PL=1
MOVL C00509 V=30.0 PL=1
MOVL C00510 V=30.0 PL=1
MOVL C00511 V=30.0 PL=1
MOVL C00512 V=30.0 PL=1
MOVL C00513 V=30.0 PL=1
MOVL C00514 V=130.0 PL=1
MOVL C00515 V=130.0 PL=1
MOVL C00516 V=20.0 PL=1
MOVL C00517 V=130.0 PL=1
MOVL C00518 V=130.0 PL=1
MOVL C00519 V=60.0 PL=1
MOVL C00520 V=60.0 PL=1
MOVL C00521 V=60.0 PL=1
MOVL C00522 V=60.0 PL=1
MOVL C00523 V=130.0 PL=1
MOVL C00524 V=30.0 PL=1
MOVL C00525 V=30.0 PL=1
MOVL C00526 V=30.0 PL=1
MOVL C00527 V=30.0 PL=1
MOVL C00528 V=30.0 PL=1
MOVL C00529 V=30.0 PL=1
MOVL C00530 V=30.0 PL=1
MOVL C00531 V=30.0 PL=1
MOVL C00532 V=130.0 PL=1
MOVL C00533 V=130.0 PL=1
MOVL C00534 V=20.0 PL=1
MOVL C00535 V=130.0 PL=1
MOVL C00536 V=130.0 PL=1
MOVL C00537 V=60.0 PL=1
MOVL C00538 V=60.0 PL=1
MOVL C00539 V=60.0 PL=1
MOVL C00540 V=60.0 PL=1
MOVL C00541 V=130.0 PL=1
MOVL C00542 V=30.0 PL=1
MOVL C00543 V=30.0 PL=1
MOVL C00544 V=30.0 PL=1
MOVL C00545 V=30.0 PL=1
MOVL C00546 V=30.0 PL=1
MOVL C00547 V=30.0 PL=1
MOVL C00548 V=30.0 PL=1
MOVL C00549 V=30.0 PL=1
MOVL C00550 V=130.0 PL=1
MOVL C00551 V=130.0 PL=1
MOVL C00552 V=20.0 PL=1
MOVL C00553 V=130.0 PL=1
MOVL C00554 V=130.0 PL=1
MOVL C00555 V=60.0 PL=1
MOVL C00556 V=60.0 PL=1
MOVL C00557 V=60.0 PL=1
MOVL C00558 V=60.0 PL=1
MOVL C00559 V=130.0 PL=1
MOVL C00560 V=30.0 PL=1
MOVL C00561 V=30.0 PL=1
MOVL C00562 V=30.0 PL=1
MOVL C00563 V=30.0 PL=1
MOVL C00564 V=30.0 PL=1
MOVL C00565 V=30.0 PL=1
MOVL C00566 V=30.0 PL=1
MOVL C00567 V=30.0 PL=1
MOVL C00568 V=130.0 PL=1
MOVL C00569 V=130.0 PL=1
MOVL C00570 V=20.0 PL=1
MOVL C00571 V=130.0 PL=1
MOVL C00572 V=130.0 PL=1
MOVL C00573 V=60.0 PL=1
MOVL C00574 V=60.0 PL=1
MOVL C00575 V=60.0 PL=1
MOVL C00576 V=60.0 PL=1
MOVL C00577 V=130.0 PL=1
MOVL C00578 V=30.0 PL=1
MOVL C00579 V=30.0 PL=1
MOVL C00580 V=30.0 PL=1
MOVL C00581 V=30.0 PL=1
MOVL C00582 V=30.0 PL=1
MOVL C00583 V=30.0 PL=1
MOVL C00584 V=30.0 PL=1
MOVL C00585 V=30.0 PL=1
MOVL C00586 V=130.0 PL=1
MOVL C00587 V=130.0 PL=1
MOVL C00588 V=20.0 PL=1
MOVL C00589 V=130.0 PL=1
MOVL C00590 V=130.0 PL=1
MOVL C00591 V=60.0 PL=1
MOVL C00592 V=60.0 PL=1
MOVL C00593 V=60.0 PL=1
MOVL C00594 V=60.0 PL=1
MOVL C00595 V=130.0 PL=1
MOVL C00596 V=30.0 PL=1
MOVL C00597 V=30.0 PL=1
MOVL C00598 V=30.0 PL=1
MOVL C00599 V=30.0 PL=1
MOVL C00600 V=30.0 PL=1
MOVL C00601 V=30.0 PL=1
MOVL C00602 V=30.0 PL=1
MOVL C00603 V=30.0 PL=1
MOVL C00604 V=130.0 PL=1
MOVL C00605 V=130.0 PL=1
MOVL C00606 V=20.0 PL=1
MOVL C00607 V=130.0 PL=1
MOVL C00608 V=130.0 PL=1
MOVL C00609 V=60.0 PL=1
MOVL C00610 V=60.0 PL=1
MOVL C00611 V=60.0 PL=1
MOVL C00612 V=60.0 PL=1
MOVL C00613 V=130.0 PL=1
MOVL C00614 V=30.0 PL=1
MOVL C00615 V=30.0 PL=1
MOVL C00616 V=30.0 PL=1
MOVL C00617 V=30.0 PL=1
MOVL C00618 V=30.0 PL=1
MOVL C00619 V=30.0 PL=1
MOVL C00620 V=30.0 PL=1
MOVL C00621 V=30.0 PL=1
MOVL C00622 V=130.0 PL=1
MOVL C00623 V=130.0 PL=1
MOVL C00624 V=20.0 PL=1
MOVL C00625 V=130.0 PL=1
MOVL C00626 V=130.0 PL=1
MOVL C00627 V=60.0 PL=1
MOVL C00628 V=60.0 PL=1
MOVL C00629 V=60.0 PL=1
MOVL C00630 V=60.0 PL=1
MOVL C00631 V=130.0 PL=1
MOVL C00632 V=30.0 PL=1
MOVL C00633 V=30.0 PL=1
MOVL C00634 V=30.0 PL=1
MOVL C00635 V=30.0 PL=1
MOVL C00636 V=30.0 PL=1
MOVL C00637 V=30.0 PL=1
MOVL C00638 V=30.0 PL=1
MOVL C00639 V=30.0 PL=1
MOVL C00640 V=130.0 PL=1
MOVL C00641 V=130.0 PL=1
MOVL C00642 V=20.0 PL=1
MOVL C00643 V=130.0 PL=1
MOVL C00644 V=130.0 PL=1
MOVL C00645 V=60.0 PL=1
MOVL C00646 V=60.0 PL=1
MOVL C00647 V=60.0 PL=1
MOVL C00648 V=60.0 PL=1
MOVL C00649 V=130.0 PL=1
MOVL C00650 V=30.0 PL=1
MOVL C00651 V=30.0 PL=1
MOVL C00652 V=30.0 PL=1
MOVL C00653 V=30.0 PL=1
MOVL C00654 V=30.0 PL=1
MOVL C00655 V=30.0 PL=1
MOVL C00656 V=30.0 PL=1
MOVL C00657 V=30.0 PL=1
MOVL C00658 V=130.0 PL=1
MOVL C00659 V=130.0 PL=1
MOVL C00660 V=20.0 PL=1
MOVL C00661 V=130.0 PL=1
MOVL C00662 V=130.0 PL=1
MOVL C00663 V=60.0 PL=1
MOVL C00664 V=60.0 PL=1
MOVL C00665 V=60.0 PL=1
MOVL C00666 V=60.0 PL=1
MOVL C00667 V=130.0 PL=1
MOVL C00668 V=30.0 PL=1
MOVL C00669 V=30.0 PL=1
MOVL C00670 V=30.0 PL=1
MOVL C00671 V=30.0 PL=1
MOVL C00672 V=30.0 PL=1
MOVL C00673 V=30.0 PL=1
MOVL C00674 V=30.0 PL=1
MOVL C00675 V=30.0 PL=1
MOVL C00676 V=130.0 PL=1
MOVL C00677 V=130.0 PL=1
MOVL C00678 V=20.0 PL=1
MOVL C00679 V=130.0 PL=1
MOVL C00680 V=130.0 PL=1
MOVL C00681 V=60.0 PL=1
MOVL C00682 V=60.0 PL=1
MOVL C00683 V=60.0 PL=1
MOVL C00684 V=60.0 PL=1
MOVL C00685 V=130.0 PL=1
MOVL C00686 V=30.0 PL=1
MOVL C00687 V=30.0 PL=1
MOVL C00688 V=30.0 PL=1
MOVL C00689 V=30.0 PL=1
MOVL C00690 V=30.0 PL=1
MOVL C00691 V=30.0 PL=1
MOVL C00692 V=30.0 PL=1
MOVL C00693 V=30.0 PL=1
MOVL C00694 V=130.0 PL=1
MOVL C00695 V=130.0 PL=1
MOVL C00696 V=20.0 PL=1
MOVL C00697 V=130.0 PL=1
MOVL C00698 V=130.0 PL=1
MOVL C00699 V=60.0 PL=1
MOVL C00700 V=60.0 PL=1
MOVL C00701 V=60.0 PL=1
MOVL C00702 V=60.0 PL=1
MOVL C00703 V=130.0 PL=1
MOVL C00704 V=30.0 PL=1
MOVL C00705 V=30.0 PL=1
MOVL C00706 V=30.0 PL=1
MOVL C00707 V=30.0 PL=1
MOVL C00708 V=30.0 PL=1
MOVL C00709 V=30.0 PL=1
MOVL C00710 V=30.0 PL=1
MOVL C00711 V=30.0 PL=1
MOVL C00712 V=130.0 PL=1
MOVL C00713 V=130.0 PL=1
MOVL C00714 V=20.0 PL=1
MOVL C00715 V=130.0 PL=1
MOVL C00716 V=130.0 PL=1
MOVL C00717 V=60.0 PL=1
MOVL C00718 V=60.0 PL=1
MOVL C00719 V=60.0 PL=1
MOVL C00720 V=60.0 PL=1
MOVL C00721 V=130.0 PL=1
MOVL C00722 V=30.0 PL=1
MOVL C00723 V=30.0 PL=1
MOVL C00724 V=30.0 PL=1
MOVL C00725 V=30.0 PL=1
MOVL C00726 V=30.0 PL=1
MOVL C00727 V=30.0 PL=1
MOVL C00728 V=30.0 PL=1
MOVL C00729 V=30.0 PL=1
MOVL C00730 V=130.0 PL=1
MOVL C00731 V=130.0 PL=1
MOVL C00732 V=20.0 PL=1
MOVL C00733 V=130.0 PL=1
MOVL C00734 V=130.0 PL=1
MOVL C00735 V=60.0 PL=1
MOVL C00736 V=60.0 PL=1
MOVL C00737 V=60.0 PL=1
MOVL C00738 V=60.0 PL=1
MOVL C00739 V=130.0 PL=1
MOVL C00740 V=30.0 PL=1
MOVL C00741 V=30.0 PL=1
MOVL C00742 V=30.0 PL=1
MOVL C00743 V=30.0 PL=1
MOVL C00744 V=30.0 PL=1
MOVL C00745 V=30.0 PL=1
MOVL C00746 V=30.0 PL=1
MOVL C00747 V=30.0 PL=1
MOVL C00748 V=130.0 PL=1
MOVL C00749 V=130.0 PL=1
MOVL C00750 V=20.0 PL=1
MOVL C00751 V=130.0 PL=1
MOVL C00752 V=130.0 PL=1
MOVL C00753 V=60.0 PL=1
MOVL C00754 V=60.0 PL=1
MOVL C00755 V=60.0 PL=1
MOVL C00756 V=60.0 PL=1
MOVL C00757 V=130.0 PL=1
MOVL C00758 V=30.0 PL=1
MOVL C00759 V=30.0 PL=1
MOVL C00760 V=30.0 PL=1
MOVL C00761 V=30.0 PL=1
MOVL C00762 V=30.0 PL=1
MOVL C00763 V=30.0 PL=1
MOVL C00764 V=30.0 PL=1
MOVL C00765 V=30.0 PL=1
MOVL C00766 V=130.0 PL=1
MOVL C00767 V=130.0 PL=1
MOVL C00768 V=20.0 PL=1
MOVL C00769 V=130.0 PL=1
MOVL C00770 V=130.0 PL=1
MOVL C00771 V=60.0 PL=1
MOVL C00772 V=60.0 PL=1
MOVL C00773 V=60.0 PL=1
MOVL C00774 V=60.0 PL=1
MOVL C00775 V=130.0 PL=1
MOVL C00776 V=30.0 PL=1
MOVL C00777 V=30.0 PL=1
MOVL C00778 V=30.0 PL=1
MOVL C00779 V=30.0 PL=1
MOVL C00780 V=30.0 PL=1
MOVL C00781 V=30.0 PL=1
MOVL C00782 V=30.0 PL=1
MOVL C00783 V=30.0 PL=1
MOVL C00784 V=130.0 PL=1
MOVL C00785 V=130.0 PL=1
MOVL C00786 V=20.0 PL=1
MOVL C00787 V=130.0 PL=1
MOVL C00788 V=130.0 PL=1
MOVL C00789 V=60.0 PL=1
MOVL C00790 V=60.0 PL=1
MOVL C00791 V=60.0 PL=1
MOVL C00792 V=60.0 PL=1
MOVL C00793 V=130.0 PL=1
MOVL C00794 V=30.0 PL=1
MOVL C00795 V=30.0 PL=1
MOVL C00796 V=30.0 PL=1
MOVL C00797 V=30.0 PL=1
MOVL C00798 V=30.0 PL=1
MOVL C00799 V=30.0 PL=1
MOVL C00800 V=30.0 PL=1
MOVL C00801 V=30.0 PL=1
MOVL C00802 V=130.0 PL=1
MOVL C00803 V=130.0 PL=1
MOVL C00804 V=20.0 PL=1
MOVL C00805 V=130.0 PL=1
MOVL C00806 V=130.0 PL=1
MOVL C00807 V=60.0 PL=1
MOVL C00808 V=60.0 PL=1
MOVL C00809 V=60.0 PL=1
MOVL C00810 V=60.0 PL=1
MOVL C00811 V=130.0 PL=1
MOVL C00812 V=30.0 PL=1
MOVL C00813 V=30.0 PL=1
MOVL C00814 V=30.0 PL=1
MOVL C00815 V=30.0 PL=1
MOVL C00816 V=30.0 PL=1
MOVL C00817 V=30.0 PL=1
MOVL C00818 V=30.0 PL=1
MOVL C00819 V=30.0 PL=1
MOVL C00820 V=130.0 PL=1
MOVL C00821 V=130.0 PL=1
MOVL C00822 V=20.0 PL=1
MOVL C00823 V=130.0 PL=1
MOVL C00824 V=130.0 PL=1
MOVL C00825 V=60.0 PL=1
MOVL C00826 V=60.0 PL=1
MOVL C00827 V=60.0 PL=1
MOVL C00828 V=60.0 PL=1
MOVL C00829 V=130.0 PL=1
MOVL C00830 V=30.0 PL=1
MOVL C00831 V=30.0 PL=1
MOVL C00832 V=30.0 PL=1
MOVL C00833 V=30.0 PL=1
MOVL C00834 V=30.0 PL=1
MOVL C00835 V=30.0 PL=1
MOVL C00836 V=30.0 PL=1
MOVL C00837 V=30.0 PL=1
MOVL C00838 V=130.0 PL=1
MOVL C00839 V=130.0 PL=1
MOVL C00840 V=20.0 PL=1
MOVL C00841 V=130.0 PL=1
MOVL C00842 V=130.0 PL=1
MOVL C00843 V=60.0 PL=1
MOVL C00844 V=60.0 PL=1
MOVL C00845 V=60.0 PL=1
MOVL C00846 V=60.0 PL=1
MOVL C00847 V=130.0 PL=1
MOVL C00848 V=30.0 PL=1
MOVL C00849 V=30.0 PL=1
MOVL C00850 V=30.0 PL=1
MOVL C00851 V=30.0 PL=1
MOVL C00852 V=30.0 PL=1
MOVL C00853 V=30.0 PL=1
MOVL C00854 V=30.0 PL=1
MOVL C00855 V=30.0 PL=1
MOVL C00856 V=130.0 PL=1
MOVL C00857 V=130.0 PL=1
MOVL C00858 V=20.0 PL=1
MOVL C00859 V=130.0 PL=1
MOVL C00860 V=130.0 PL=1
MOVL C00861 V=60.0 PL=1
MOVL C00862 V=60.0 PL=1
MOVL C00863 V=60.0 PL=1
MOVL C00864 V=60.0 PL=1
MOVL C00865 V=130.0 PL=1
MOVL C00866 V=30.0 PL=1
MOVL C00867 V=30.0 PL=1
MOVL C00868 V=30.0 PL=1
MOVL C00869 V=30.0 PL=1
MOVL C00870 V=30.0 PL=1
MOVL C00871 V=30.0 PL=1
MOVL C00872 V=30.0 PL=1
MOVL C00873 V=30.0 PL=1
MOVL C00874 V=130.0 PL=1
MOVL C00875 V=130.0 PL=1
MOVL C00876 V=20.0 PL=1
MOVL C00877 V=130.0 PL=1
MOVL C00878 V=130.0 PL=1
MOVL C00879 V=60.0 PL=1
MOVL C00880 V=60.0 PL=1
MOVL C00881 V=60.0 PL=1
MOVL C00882 V=60.0 PL=1
MOVL C00883 V=130.0 PL=1
MOVL C00884 V=30.0 PL=1
MOVL C00885 V=30.0 PL=1
MOVL C00886 V=30.0 PL=1
MOVL C00887 V=30.0 PL=1
MOVL C00888 V=30.0 PL=1
MOVL C00889 V=30.0 PL=1
MOVL C00890 V=30.0 PL=1
MOVL C00891 V=30.0 PL=1
MOVL C00892 V=130.0 PL=1
MOVL C00893 V=130.0 PL=1
MOVL C00894 V=20.0 PL=1
MOVL C00895 V=130.0 PL=1
MOVL C00896 V=130.0 PL=1
MOVL C00897 V=60.0 PL=1
MOVL C00898 V=60.0 PL=1
MOVL C00899 V=60.0 PL=1
MOVL C00900 V=60.0 PL=1
MOVL C00901 V=130.0 PL=1
MOVL C00902 V=30.0 PL=1
MOVL C00903 V=30.0 PL=1
MOVL C00904 V=30.0 PL=1
MOVL C00905 V=30.0 PL=1
MOVL C00906 V=30.0 PL=1
MOVL C00907 V=30.0 PL=1
MOVL C00908 V=30.0 PL=1
MOVL C00909 V=30.0 PL=1
MOVL C00910 V=130.0 PL=1
MOVL C00911 V=130.0 PL=1
MOVL C00912 V=20.0 PL=1
MOVL C00913 V=130.0 PL=1
MOVL C00914 V=130.0 PL=1
MOVL C00915 V=60.0 PL=1
MOVL C00916 V=60.0 PL=1
MOVL C00917 V=60.0 PL=1
MOVL C00918 V=60.0 PL=1
MOVL C00919 V=130.0 PL=1
MOVL C00920 V=30.0 PL=1
MOVL C00921 V=30.0 PL=1
MOVL C00922 V=30.0 PL=1
MOVL C00923 V=30.0 PL=1
MOVL C00924 V=30.0 PL=1
MOVL C00925 V=30.0 PL=1
MOVL C00926 V=30.0 PL=1
MOVL C00927 V=30.0 PL=1
MOVL C00928 V=130.0 PL=1
MOVL C00929 V=130.0 PL=1
MOVL C00930 V=20.0 PL=1
MOVL C00931 V=130.0 PL=1
MOVL C00932 V=130.0 PL=1
MOVL C00933 V=60.0 PL=1
MOVL C00934 V=60.0 PL=1
MOVL C00935 V=60.0 PL=1
MOVL C00936 V=60.0 PL=1
MOVL C00937 V=130.0 PL=1
MOVL C00938 V=30.0 PL=1
MOVL C00939 V=30.0 PL=1
MOVL C00940 V=30.0 PL=1
MOVL C00941 V=30.0 PL=1
MOVL C00942 V=30.0 PL=1
MOVL C00943 V=30.0 PL=1
MOVL C00944 V=30.0 PL=1
MOVL C00945 V=30.0 PL=1
MOVL C00946 V=130.0 PL=1
MOVL C00947 V=130.0 PL=1
MOVL C00948 V=20.0 PL=1
MOVL C00949 V=130.0 PL=1
MOVL C00950 V=130.0 PL=1
MOVL C00951 V=60.0 PL=1
MOVL C00952 V=60.0 PL=1
MOVL C00953 V=60.0 PL=1
MOVL C00954 V=60.0 PL=1
MOVL C00955 V=130.0 PL=1
MOVL C00956 V=30.0 PL=1
MOVL C00957 V=30.0 PL=1
MOVL C00958 V=30.0 PL=1
MOVL C00959 V=30.0 PL=1
MOVL C00960 V=30.0 PL=1
MOVL C00961 V=30.0 PL=1
MOVL C00962 V=30.0 PL=1
MOVL C00963 V=30.0 PL=1
MOVL C00964 V=130.0 PL=1
MOVL C00965 V=130.0 PL=1
MOVL C00966 V=20.0 PL=1
MOVL C00967 V=130.0 PL=1
MOVL C00968 V=130.0 PL=1
MOVL C00969 V=60.0 PL=1
MOVL C00970 V=60.0 PL=1
MOVL C00971 V=60.0 PL=1
MOVL C00972 V=60.0 PL=1
MOVL C00973 V=130.0 PL=1
MOVL C00974 V=30.0 PL=1
MOVL C00975 V=30.0 PL=1
MOVL C00976 V=30.0 PL=1
MOVL C00977 V=30.0 PL=1
MOVL C00978 V=30.0 PL=1
MOVL C00979 V=30.0 PL=1
MOVL C00980 V=30.0 PL=1
MOVL C00981 V=30.0 PL=1
MOVL C00982 V=130.0 PL=1
MOVL C00983 V=130.0 PL=1
MOVL C00984 V=20.0 PL=1
MOVL C00985 V=130.0 PL=1
MOVL C00986 V=130.0 PL=1
MOVL C00987 V=60.0 PL=1
MOVL C00988 V=60.0 PL=1
MOVL C00989 V=60.0 PL=1
MOVL C00990 V=60.0 PL=1
MOVL C00991 V=130.0 PL=1
MOVL C00992 V=30.0 PL=1
MOVL C00993 V=30.0 PL=1
MOVL C00994 V=30.0 PL=1
MOVL C00995 V=30.0 PL=1
MOVL C00996 V=30.0 PL=1
MOVL C00997 V=30.0 PL=1
MOVL C00998 V=30.0 PL=1
MOVL C00999 V=30.0 PL=1
MOVL C01000 V=130.0 PL=1
MOVL C01001 V=130.0 PL=1
MOVL C01002 V=20.0 PL=1
MOVL C01003 V=130.0 PL=1
MOVL C01004 V=130.0 PL=1
MOVL C01005 V=60.0 PL=1
MOVL C01006 V=60.0 PL=1
MOVL C01007 V=60.0 PL=1
MOVL C01008 V=60.0 PL=1
MOVL C01009 V=130.0 PL=1
MOVL C01010 V=30.0 PL=1
MOVL C01011 V=30.0 PL=1
MOVL C01012 V=30.0 PL=1
MOVL C01013 V=30.0 PL=1
MOVL C01014 V=30.0 PL=1
MOVL C01015 V=30.0 PL=1
MOVL C01016 V=30.0 PL=1
MOVL C01017 V=30.0 PL=1
MOVL C01018 V=130.0 PL=1
MOVL C01019 V=130.0 PL=1
MOVL C01020 V=20.0 PL=1
MOVL C01021 V=130.0 PL=1
MOVL C01022 V=130.0 PL=1
MOVL C01023 V=60.0 PL=1
MOVL C01024 V=60.0 PL=1
MOVL C01025 V=60.0 PL=1
MOVL C01026 V=60.0 PL=1
MOVL C01027 V=130.0 PL=1
MOVL C01028 V=30.0 PL=1
MOVL C01029 V=30.0 PL=1
MOVL C01030 V=30.0 PL=1
MOVL C01031 V=30.0 PL=1
MOVL C01032 V=30.0 PL=1
MOVL C01033 V=30.0 PL=1
MOVL C01034 V=30.0 PL=1
MOVL C01035 V=30.0 PL=1
MOVL C01036 V=130.0 PL=1
MOVL C01037 V=130.0 PL=1
MOVL C01038 V=20.0 PL=1
MOVL C01039 V=130.0 PL=1
MOVL C01040 V=130.0 PL=1
MOVL C01041 V=60.0 PL=1
MOVL C01042 V=60.0 PL=1
MOVL C01043 V=60.0 PL=1
MOVL C01044 V=60.0 PL=1
MOVL C01045 V=130.0 PL=1
MOVL C01046 V=30.0 PL=1
MOVL C01047 V=30.0 PL=1
MOVL C01048 V=30.0 PL=1
MOVL C01049 V=30.0 PL=1
MOVL C01050 V=30.0 PL=1
MOVL C01051 V=30.0 PL=1
MOVL C01052 V=30.0 PL=1
MOVL C01053 V=30.0 PL=1
MOVL C01054 V=130.0 PL=1
MOVL C01055 V=130.0 PL=1
MOVL C01056 V=20.0 PL=1
MOVL C01057 V=130.0 PL=1
MOVL C01058 V=130.0 PL=1
MOVL C01059 V=60.0 PL=1
MOVL C01060 V=60.0 PL=1
MOVL C01061 V=60.0 PL=1
MOVL C01062 V=60.0 PL=1
MOVL C01063 V=130.0 PL=1
MOVL C01064 V=30.0 PL=1
MOVL C01065 V=30.0 PL=1
MOVL C01066 V=30.0 PL=1
MOVL C01067 V=30.0 PL=1
MOVL C01068 V=30.0 PL=1
MOVL C01069 V=30.0 PL=1
MOVL C01070 V=30.0 PL=1
MOVL C01071 V=30.0 PL=1
MOVL C01072 V=130.0 PL=1
MOVL C01073 V=130.0 PL=1
MOVL C01074 V=20.0 PL=1
MOVL C01075 V=130.0 PL=1
MOVL C01076 V=130.0 PL=1
MOVL C01077 V=60.0 PL=1
MOVL C01078 V=60.0 PL=1
MOVL C01079 V=60.0 PL=1
MOVL C01080 V=60.0 PL=1
MOVL C01081 V=130.0 PL=1
MOVL C01082 V=30.0 PL=1
MOVL C01083 V=30.0 PL=1
MOVL C01084 V=30.0 PL=1
MOVL C01085 V=30.0 PL=1
MOVL C01086 V=30.0 PL=1
MOVL C01087 V=30.0 PL=1
MOVL C01088 V=30.0 PL=1
MOVL C01089 V=30.0 PL=1
MOVL C01090 V=130.0 PL=1
MOVL C01091 V=130.0 PL=1
MOVL C01092 V=20.0 PL=1
MOVL C01093 V=130.0 PL=1
MOVL C01094 V=130.0 PL=1
MOVL C01095 V=60.0 PL=1
MOVL C01096 V=60.0 PL=1
MOVL C01097 V=60.0 PL=1
MOVL C01098 V=60.0 PL=1
MOVL C01099 V=130.0 PL=1
MOVL C01100 V=30.0 PL=1
MOVL C01101 V=30.0 PL=1
MOVL C01102 V=30.0 PL=1
MOVL C01103 V=30.0 PL=1
MOVL C01104 V=30.0 PL=1
MOVL C01105 V=30.0 PL=1
MOVL C01106 V=30.0 PL=1
MOVL C01107 V=30.0 PL=1
MOVL C01108 V=130.0 PL=1
MOVL C01109 V=130.0 PL=1
MOVL C01110 V=20.0 PL=1
MOVL C01111 V=130.0 PL=1
MOVL C01112 V=130.0 PL=1
MOVL C01113 V=60.0 PL=1
MOVL C01114 V=60.0 PL=1
MOVL C01115 V=60.0 PL=1
MOVL C01116 V=60.0 PL=1
MOVL C01117 V=130.0 PL=1
MOVL C01118 V=30.0 PL=1
MOVL C01119 V=30.0 PL=1
MOVL C01120 V=30.0 PL=1
MOVL C01121 V=30.0 PL=1
MOVL C01122 V=30.0 PL=1
MOVL C01123 V=30.0 PL=1
MOVL C01124 V=30.0 PL=1
MOVL C01125 V=30.0 PL=1
MOVL C01126 V=130.0 PL=1
MOVL C01127 V=130.0 PL=1
MOVL C01128 V=20.0 PL=1
MOVL C01129 V=130.0 PL=1
MOVL C01130 V=130.0 PL=1
MOVL C01131 V=60.0 PL=1
MOVL C01132 V=60.0 PL=1
MOVL C01133 V=60.0 PL=1
MOVL C01134 V=60.0 PL=1
MOVL C01135 V=130.0 PL=1
MOVL C01136 V=30.0 PL=1
MOVL C01137 V=30.0 PL=1
MOVL C01138 V=30.0 PL=1
MOVL C01139 V=30.0 PL=1
MOVL C01140 V=30.0 PL=1
MOVL C01141 V=30.0 PL=1
MOVL C01142 V=30.0 PL=1
MOVL C01143 V=30.0 PL=1
MOVL C01144 V=130.0 PL=1
MOVL C01145 V=130.0 PL=1
MOVL C01146 V=20.0 PL=1
MOVL C01147 V=130.0 PL=1
MOVL C01148 V=130.0 PL=1
MOVL C01149 V=60.0 PL=1
MOVL C01150 V=60.0 PL=1
MOVL C01151 V=60.0 PL=1
MOVL C01152 V=60.0 PL=1
MOVL C01153 V=130.0 PL=1
MOVL C01154 V=30.0 PL=1
MOVL C01155 V=30.0 PL=1
MOVL C01156 V=30.0 PL=1
MOVL C01157 V=30.0 PL=1
MOVL C01158 V=30.0 PL=1
MOVL C01159 V=30.0 PL=1
MOVL C01160 V=30.0 PL=1
END
